Yaskawa INFORM job: DPRINT3D16.JBI

/JOB
//NAME DPRINT3D16
//POS
///NPOS 1162,0,0,0,0,0
///TOOL 9
///POSTYPE PULSE
///PULSE
C00000=35629,41672,-114626,80977,-121328,-83417,0
C00001=36190,41299,-115490,80334,-121553,-83708,0
C00002=36154,40665,-116948,80172,-121272,-84071,0
C00003=40236,36747,-126052,74955,-121987,-86900,0
C00004=40236,36690,-126053,74971,-122014,-86869,0
C00005=36377,41178,-115654,80151,-121668,-83746,0
C00006=41048,36722,-125993,74163,-122491,-86973,0
C00007=40041,36151,-127297,75001,-121635,-87147,0
C00008=35414,40629,-116901,80893,-120814,-83936,0
C00009=36299,41132,-115758,80210,-121598,-83762,0
C00010=35683,41556,-114775,80921,-121358,-83434,0
C00011=36557,42075,-113598,80267,-122151,-83252,0
C00012=42279,36667,-126139,72897,-123156,-87194,0
C00013=39910,35322,-129213,74883,-121147,-87599,0
C00014=34311,40792,-116511,81978,-120152,-83701,0
C00015=35213,41288,-115384,81279,-120939,-83528,0
C00016=34977,41570,-114734,81585,-120890,-83333,0
C00017=35446,41838,-114126,81230,-121308,-83239,0
C00018=35629,41620,-114628,80992,-121347,-83390,0
C00019=36191,41247,-115492,80349,-121573,-83680,0
C00020=36155,40612,-116951,80186,-121292,-84043,0
C00021=40236,36690,-126053,74971,-122014,-86869,0
C00022=40237,36632,-126055,74988,-122040,-86840,0
C00023=36378,41126,-115657,80166,-121688,-83719,0
C00024=41048,36664,-125996,74179,-122518,-86943,0
C00025=40042,36093,-127299,75017,-121661,-87117,0
C00026=35414,40576,-116904,80907,-120834,-83907,0
C00027=36300,41080,-115760,80225,-121617,-83734,0
C00028=35684,41505,-114777,80936,-121377,-83406,0
C00029=36558,42025,-113599,80281,-122170,-83225,0
C00030=42279,36610,-126142,72914,-123184,-87165,0
C00031=39910,35263,-129216,74898,-121175,-87568,0
C00032=34311,40739,-116513,81992,-120171,-83672,0
C00033=35213,41236,-115387,81294,-120959,-83500,0
C00034=34977,41518,-114736,81599,-120908,-83306,0
C00035=35446,41787,-114128,81244,-121328,-83211,0
C00036=35629,41569,-114630,81006,-121366,-83362,0
C00037=36191,41196,-115494,80363,-121592,-83653,0
C00038=36155,40560,-116952,80201,-121312,-84015,0
C00039=40237,36632,-126055,74988,-122040,-86840,0
C00040=40237,36575,-126058,75004,-122067,-86810,0
C00041=36378,41074,-115658,80180,-121707,-83691,0
C00042=41049,36607,-125997,74196,-122546,-86914,0
C00043=40042,36034,-127300,75033,-121689,-87086,0
C00044=35414,40524,-116905,80921,-120853,-83879,0
C00045=36300,41029,-115761,80240,-121637,-83706,0
C00046=35684,41454,-114778,80950,-121396,-83379,0
C00047=36558,41974,-113601,80296,-122190,-83197,0
C00048=42279,36552,-126143,72931,-123212,-87135,0
C00049=39911,35204,-129217,74914,-121201,-87537,0
C00050=34311,40687,-116514,82006,-120189,-83644,0
C00051=35214,41184,-115388,81308,-120977,-83472,0
C00052=34978,41467,-114738,81613,-120927,-83278,0
C00053=35447,41736,-114129,81258,-121346,-83184,0
C00054=35630,41518,-114631,81020,-121385,-83334,0
C00055=36191,41144,-115496,80378,-121612,-83625,0
C00056=36155,40507,-116953,80215,-121331,-83987,0
C00057=40237,36575,-126058,75004,-122067,-86810,0
C00058=40238,36518,-126059,75020,-122093,-86780,0
C00059=36378,41022,-115659,80195,-121727,-83663,0
C00060=41049,36550,-125999,74212,-122572,-86884,0
C00061=40042,35976,-127302,75049,-121715,-87056,0
C00062=35415,40471,-116907,80935,-120873,-83851,0
C00063=36300,40977,-115762,80254,-121657,-83679,0
C00064=35684,41402,-114780,80965,-121415,-83351,0
C00065=36558,41923,-113603,80311,-122209,-83170,0
C00066=42280,36495,-126145,72948,-123241,-87106,0
C00067=39911,35144,-129219,74930,-121229,-87507,0
C00068=34312,40635,-116515,82019,-120207,-83616,0
C00069=35214,41133,-115390,81322,-120996,-83444,0
C00070=34978,41415,-114739,81627,-120946,-83250,0
C00071=35447,41685,-114131,81273,-121365,-83157,0
C00072=35630,41466,-114633,81035,-121404,-83307,0
C00073=36192,41092,-115497,80393,-121631,-83597,0
C00074=36156,40455,-116955,80230,-121352,-83959,0
C00075=40238,36518,-126059,75020,-122093,-86780,0
C00076=40238,36460,-126060,75036,-122120,-86750,0
C00077=36379,40971,-115661,80210,-121746,-83635,0
C00078=41050,36492,-126000,74229,-122600,-86854,0
C00079=40043,35918,-127303,75065,-121742,-87026,0
C00080=35415,40419,-116908,80950,-120892,-83823,0
C00081=36301,40925,-115765,80269,-121677,-83651,0
C00082=35685,41351,-114781,80979,-121434,-83323,0
C00083=36559,41872,-113604,80326,-122228,-83142,0
C00084=42280,36438,-126146,72965,-123269,-87076,0
C00085=39912,35085,-129220,74946,-121257,-87476,0
C00086=34312,40583,-116517,82033,-120226,-83588,0
C00087=35214,41081,-115391,81336,-121015,-83416,0
C00088=34978,41364,-114741,81641,-120965,-83223,0
C00089=35447,41634,-114132,81287,-121383,-83129,0
C00090=35630,41415,-114634,81049,-121422,-83279,0
C00091=36192,41040,-115498,80408,-121651,-83569,0
C00092=36156,40403,-116956,80245,-121372,-83930,0
C00093=40238,36460,-126060,75036,-122120,-86750,0
C00094=40238,36403,-126062,75052,-122146,-86720,0
C00095=36379,40919,-115663,80225,-121767,-83607,0
C00096=41050,36435,-126001,74245,-122626,-86824,0
C00097=40043,35860,-127305,75081,-121769,-86996,0
C00098=35415,40367,-116909,80964,-120912,-83795,0
C00099=36301,40873,-115766,80284,-121697,-83623,0
C00100=35685,41300,-114783,80994,-121453,-83296,0
C00101=36559,41821,-113605,80341,-122247,-83115,0
C00102=42281,36380,-126149,72982,-123297,-87046,0
C00103=39912,35026,-129223,74962,-121284,-87445,0
C00104=34312,40531,-116519,82047,-120244,-83560,0
C00105=35215,41030,-115392,81351,-121034,-83388,0
C00106=34979,41313,-114742,81656,-120983,-83195,0
C00107=35448,41583,-114134,81302,-121401,-83101,0
C00108=35631,41364,-114636,81064,-121442,-83251,0
C00109=36192,40989,-115500,80422,-121670,-83542,0
C00110=36156,40350,-116958,80260,-121392,-83902,0
C00111=40238,36403,-126062,75052,-122146,-86720,0
C00112=40239,36346,-126064,75069,-122172,-86690,0
C00113=36379,40867,-115664,80240,-121786,-83579,0
C00114=41051,36378,-126003,74262,-122654,-86795,0
C00115=40044,35802,-127307,75097,-121796,-86965,0
C00116=35416,40315,-116910,80979,-120931,-83767,0
C00117=36301,40822,-115767,80299,-121716,-83595,0
C00118=35685,41249,-114784,81008,-121471,-83268,0
C00119=36559,41771,-113607,80356,-122267,-83088,0
C00120=42281,36323,-126150,72999,-123325,-87017,0
C00121=39912,34966,-129224,74978,-121312,-87414,0
C00122=34312,40479,-116520,82061,-120263,-83532,0
C00123=35215,40978,-115394,81365,-121052,-83361,0
C00124=34979,41262,-114744,81670,-121001,-83167,0
C00125=35448,41532,-114135,81316,-121421,-83074,0
C00126=35631,41313,-114637,81078,-121460,-83224,0
C00127=36193,40937,-115502,80437,-121690,-83514,0
C00128=36157,40298,-116959,80274,-121412,-83874,0
C00129=40239,36346,-126064,75069,-122172,-86690,0
C00130=40239,36289,-126065,75085,-122199,-86660,0
C00131=36380,40816,-115665,80255,-121806,-83551,0
C00132=41051,36321,-126004,74279,-122682,-86764,0
C00133=40044,35744,-127308,75114,-121822,-86935,0
C00134=35416,40262,-116912,80993,-120950,-83738,0
C00135=36302,40770,-115768,80314,-121736,-83567,0
C00136=35685,41197,-114785,81023,-121491,-83240,0
C00137=36560,41720,-113608,80371,-122286,-83060,0
C00138=42281,36266,-126151,73016,-123354,-86987,0
C00139=39913,34907,-129225,74994,-121339,-87383,0
C00140=34313,40427,-116521,82075,-120281,-83503,0
C00141=35215,40927,-115395,81379,-121072,-83333,0
C00142=34979,41211,-114745,81684,-121020,-83139,0
C00143=35448,41481,-114136,81331,-121439,-83046,0
C00144=35631,41262,-114638,81093,-121480,-83196,0
C00145=36193,40886,-115503,80452,-121709,-83486,0
C00146=36157,40246,-116961,80289,-121431,-83846,0
C00147=40239,36289,-126065,75085,-122199,-86660,0
C00148=40240,36231,-126066,75101,-122225,-86630,0
C00149=36380,40764,-115666,80270,-121825,-83524,0
C00150=41051,36264,-126005,74295,-122708,-86735,0
C00151=40044,35686,-127309,75130,-121850,-86905,0
C00152=35416,40210,-116913,81007,-120969,-83710,0
C00153=36302,40718,-115769,80329,-121755,-83539,0
C00154=35686,41146,-114787,81037,-121511,-83212,0
C00155=36560,41669,-113609,80387,-122306,-83033,0
C00156=42282,36209,-126152,73033,-123383,-86957,0
C00157=39913,34848,-129226,75010,-121367,-87352,0
C00158=34313,40375,-116522,82089,-120299,-83475,0
C00159=35216,40875,-115396,81394,-121090,-83305,0
C00160=34980,41159,-114746,81698,-121038,-83112,0
C00161=35449,41430,-114137,81345,-121458,-83019,0
C00162=35632,41210,-114639,81108,-121498,-83168,0
C00163=36193,40834,-115504,80467,-121729,-83458,0
C00164=36157,40194,-116962,80304,-121452,-83818,0
C00165=40240,36231,-126066,75101,-122225,-86630,0
C00166=40240,36174,-126067,75118,-122252,-86600,0
C00167=36380,40713,-115667,80285,-121845,-83495,0
C00168=41052,36207,-126006,74312,-122736,-86705,0
C00169=40045,35629,-127310,75146,-121876,-86874,0
C00170=35417,40158,-116914,81022,-120989,-83682,0
C00171=36302,40667,-115771,80344,-121775,-83511,0
C00172=35686,41095,-114788,81052,-121529,-83184,0
C00173=36560,41619,-113610,80402,-122324,-83005,0
C00174=42282,36152,-126153,73051,-123410,-86927,0
C00175=39914,34789,-129227,75027,-121394,-87321,0
C00176=34314,40323,-116523,82102,-120318,-83447,0
C00177=35216,40824,-115397,81408,-121110,-83276,0
C00178=34980,41108,-114747,81713,-121057,-83084,0
C00179=35449,41379,-114138,81360,-121476,-82991,0
C00180=35632,41159,-114640,81122,-121517,-83141,0
C00181=36194,40783,-115505,80482,-121748,-83430,0
C00182=36158,40142,-116962,80319,-121471,-83789,0
C00183=40240,36174,-126067,75118,-122252,-86600,0
C00184=40240,36117,-126068,75134,-122278,-86570,0
C00185=36381,40661,-115668,80300,-121866,-83467,0
C00186=41052,36150,-126007,74329,-122763,-86674,0
C00187=40045,35571,-127311,75162,-121902,-86844,0
C00188=35417,40106,-116915,81036,-121008,-83654,0
C00189=36303,40615,-115772,80359,-121796,-83483,0
C00190=35687,41044,-114789,81067,-121548,-83156,0
C00191=36561,41568,-113611,80417,-122344,-82978,0
C00192=42283,36095,-126154,73068,-123439,-86897,0
C00193=39914,34730,-129228,75043,-121422,-87290,0
C00194=34314,40271,-116524,82116,-120336,-83419,0
C00195=35216,40773,-115398,81422,-121128,-83249,0
C00196=34980,41057,-114748,81727,-121075,-83056,0
C00197=35449,41328,-114139,81374,-121496,-82963,0
C00198=35632,41108,-114641,81137,-121536,-83113,0
C00199=36194,40732,-115506,80497,-121768,-83402,0
C00200=36158,40089,-116963,80334,-121492,-83761,0
C00201=40240,36117,-126068,75134,-122278,-86570,0
C00202=40241,36060,-126069,75151,-122305,-86540,0
C00203=36381,40610,-115669,80315,-121885,-83439,0
C00204=41053,36093,-126008,74346,-122790,-86645,0
C00205=40046,35513,-127313,75179,-121930,-86813,0
C00206=35417,40054,-116916,81051,-121028,-83625,0
C00207=36303,40564,-115773,80374,-121815,-83455,0
C00208=35687,40993,-114789,81082,-121567,-83128,0
C00209=36561,41518,-113612,80432,-122363,-82950,0
C00210=42283,36037,-126155,73085,-123468,-86868,0
C00211=39914,34671,-129229,75059,-121450,-87259,0
C00212=34314,40219,-116526,82130,-120355,-83390,0
C00213=35217,40721,-115399,81437,-121146,-83221,0
C00214=34981,41006,-114749,81741,-121093,-83028,0
C00215=35449,41278,-114140,81389,-121514,-82935,0
C00216=35633,41057,-114642,81152,-121555,-83085,0
C00217=36194,40680,-115506,80512,-121788,-83374,0
C00218=36158,40037,-116964,80348,-121512,-83733,0
C00219=40241,36060,-126069,75151,-122305,-86540,0
C00220=40241,36003,-126069,75167,-122331,-86510,0
C00221=36381,40558,-115669,80330,-121905,-83412,0
C00222=41053,36036,-126010,74363,-122817,-86615,0
C00223=40046,35455,-127313,75195,-121956,-86783,0
C00224=35418,40002,-116917,81065,-121047,-83597,0
C00225=36303,40512,-115773,80389,-121835,-83427,0
C00226=35687,40942,-114790,81096,-121586,-83101,0
C00227=36561,41467,-113613,80447,-122383,-82922,0
C00228=42284,35980,-126155,73103,-123495,-86837,0
C00229=39915,34612,-129229,75075,-121477,-87228,0
C00230=34314,40167,-116526,82144,-120373,-83362,0
C00231=35217,40670,-115400,81451,-121166,-83193,0
C00232=34981,40955,-114750,81756,-121112,-83000,0
C00233=35450,41227,-114141,81404,-121532,-82907,0
C00234=35633,41006,-114643,81166,-121574,-83057,0
C00235=36195,40629,-115507,80527,-121807,-83346,0
C00236=36159,39985,-116966,80363,-121531,-83705,0
C00237=40241,36003,-126069,75167,-122331,-86510,0
C00238=40242,35946,-126070,75184,-122357,-86479,0
C00239=36382,40507,-115671,80345,-121924,-83383,0
C00240=41053,35979,-126011,74380,-122845,-86584,0
C00241=40046,35397,-127314,75212,-121983,-86752,0
C00242=35418,39950,-116917,81080,-121067,-83568,0
C00243=36304,40461,-115774,80404,-121854,-83399,0
C00244=35688,40891,-114791,81111,-121605,-83073,0
C00245=36562,41417,-113614,80462,-122402,-82895,0
C00246=42284,35923,-126157,73120,-123524,-86808,0
C00247=39915,34553,-129231,75092,-121505,-87197,0
C00248=34315,40116,-116527,82158,-120391,-83333,0
C00249=35217,40619,-115400,81466,-121184,-83164,0
C00250=34981,40904,-114750,81770,-121130,-82972,0
C00251=35450,41176,-114142,81418,-121551,-82880,0
C00252=35633,40956,-114644,81181,-121593,-83029,0
C00253=36195,40577,-115509,80542,-121827,-83318,0
C00254=36159,39933,-116966,80378,-121552,-83676,0
C00255=40242,35946,-126070,75184,-122357,-86479,0
C00256=40242,35889,-126072,75200,-122385,-86449,0
C00257=36382,40456,-115672,80360,-121945,-83355,0
C00258=41054,35922,-126011,74397,-122871,-86554,0
C00259=40047,35340,-127315,75228,-122010,-86721,0
C00260=35418,39898,-116919,81095,-121087,-83540,0
C00261=36304,40409,-115775,80419,-121874,-83370,0
C00262=35688,40840,-114792,81126,-121624,-83045,0
C00263=36562,41366,-113614,80478,-122421,-82867,0
C00264=42284,35866,-126158,73137,-123553,-86778,0
C00265=39916,34494,-129232,75108,-121532,-87165,0
C00266=34315,40064,-116528,82172,-120410,-83305,0
C00267=35218,40567,-115402,81481,-121203,-83137,0
C00268=34982,40853,-114751,81784,-121149,-82944,0
C00269=35450,41126,-114142,81433,-121569,-82852,0
C00270=35634,40905,-114644,81196,-121612,-83001,0
C00271=36195,40526,-115509,80557,-121846,-83290,0
C00272=36159,39881,-116967,80393,-121571,-83648,0
C00273=40242,35889,-126072,75200,-122385,-86449,0
C00274=40242,35833,-126072,75217,-122411,-86419,0
C00275=36383,40404,-115672,80375,-121964,-83327,0
C00276=41054,35865,-126012,74413,-122899,-86524,0
C00277=40047,35282,-127315,75245,-122037,-86691,0
C00278=35419,39846,-116919,81109,-121105,-83511,0
C00279=36304,40358,-115775,80434,-121894,-83343,0
C00280=35688,40789,-114792,81141,-121643,-83017,0
C00281=36562,41316,-113615,80493,-122440,-82839,0
C00282=42285,35809,-126158,73155,-123580,-86748,0
C00283=39916,34435,-129232,75124,-121560,-87135,0
C00284=34315,40012,-116528,82187,-120428,-83277,0
C00285=35218,40516,-115402,81495,-121222,-83108,0
C00286=34982,40803,-114752,81799,-121167,-82916,0
C00287=35451,41075,-114143,81448,-121589,-82824,0
C00288=35634,40854,-114645,81211,-121630,-82973,0
C00289=36196,40475,-115510,80572,-121866,-83262,0
C00290=36160,39830,-116968,80408,-121592,-83619,0
C00291=40242,35833,-126072,75217,-122411,-86419,0
C00292=40243,35776,-126072,75234,-122438,-86388,0
C00293=36383,40353,-115672,80390,-121984,-83299,0
C00294=41055,35808,-126012,74431,-122926,-86495,0
C00295=40048,35224,-127315,75261,-122063,-86661,0
C00296=35419,39794,-116920,81124,-121124,-83483,0
C00297=36305,40307,-115775,80449,-121914,-83314,0
C00298=35688,40738,-114793,81156,-121662,-82989,0
C00299=36563,41266,-113615,80508,-122460,-82812,0
C00300=42285,35753,-126158,73172,-123609,-86718,0
C00301=39917,34376,-129233,75141,-121588,-87103,0
C00302=34316,39960,-116528,82201,-120446,-83248,0
C00303=35218,40465,-115403,81510,-121241,-83080,0
C00304=34982,40752,-114752,81813,-121185,-82888,0
C00305=35451,41024,-114143,81462,-121607,-82797,0
C00306=35634,40803,-114646,81226,-121650,-82945,0
C00307=36196,40424,-115510,80587,-121885,-83234,0
C00308=36160,39778,-116968,80423,-121612,-83591,0
C00309=40243,35776,-126072,75234,-122438,-86388,0
C00310=40243,35719,-126073,75250,-122464,-86358,0
C00311=36383,40302,-115673,80406,-122004,-83271,0
C00312=41055,35751,-126012,74448,-122953,-86464,0
C00313=40048,35167,-127316,75278,-122091,-86630,0
C00314=35419,39743,-116920,81139,-121144,-83455,0
C00315=36305,40255,-115776,80464,-121933,-83286,0
C00316=35689,40687,-114793,81170,-121681,-82961,0
C00317=36563,41215,-113616,80524,-122479,-82784,0
C00318=42286,35696,-126159,73190,-123638,-86688,0
C00319=39917,34317,-129233,75157,-121615,-87072,0
C00320=34316,39909,-116529,82215,-120465,-83220,0
C00321=35219,40414,-115403,81524,-121260,-83052,0
C00322=34983,40701,-114752,81828,-121204,-82860,0
C00323=35451,40974,-114144,81477,-121625,-82769,0
C00324=35635,40752,-114646,81240,-121668,-82917,0
C00325=36196,40373,-115511,80602,-121905,-83206,0
C00326=36161,39726,-116968,80438,-121631,-83562,0
C00327=40243,35719,-126073,75250,-122464,-86358,0
C00328=40244,35662,-126073,75267,-122491,-86328,0
C00329=36383,40251,-115673,80421,-122023,-83243,0
C00330=41055,35695,-126013,74465,-122980,-86434,0
C00331=40049,35109,-127316,75294,-122117,-86599,0
C00332=35420,39691,-116920,81153,-121164,-83426,0
C00333=36306,40204,-115776,80480,-121953,-83258,0
C00334=35689,40637,-114793,81185,-121700,-82933,0
C00335=36563,41165,-113616,80539,-122499,-82756,0
C00336=42286,35639,-126159,73208,-123665,-86658,0
C00337=39917,34258,-129233,75174,-121643,-87041,0
C00338=34316,39857,-116529,82229,-120483,-83191,0
C00339=35219,40363,-115403,81539,-121278,-83024,0
C00340=34983,40650,-114753,81843,-121222,-82832,0
C00341=35452,40923,-114144,81492,-121644,-82741,0
C00342=35635,40702,-114646,81255,-121688,-82889,0
C00343=36197,40322,-115511,80617,-121925,-83178,0
C00344=36161,39674,-116969,80454,-121652,-83534,0
C00345=40244,35662,-126073,75267,-122491,-86328,0
C00346=40244,35605,-126073,75284,-122517,-86298,0
C00347=36384,40199,-115673,80436,-122044,-83214,0
C00348=41056,35638,-126013,74482,-123008,-86403,0
C00349=40049,35052,-127316,75311,-122145,-86568,0
C00350=35420,39639,-116920,81168,-121183,-83398,0
C00351=36306,40153,-115776,80495,-121973,-83230,0
C00352=35689,40586,-114794,81200,-121719,-82905,0
C00353=36564,41115,-113616,80555,-122518,-82729,0
C00354=42286,35582,-126159,73225,-123694,-86628,0
C00355=39918,34200,-129234,75190,-121670,-87009,0
C00356=34317,39806,-116529,82243,-120502,-83163,0
C00357=35219,40312,-115404,81554,-121297,-82996,0
C00358=34983,40599,-114753,81857,-121241,-82804,0
C00359=35452,40873,-114144,81507,-121663,-82712,0
C00360=35635,40651,-114647,81270,-121706,-82861,0
C00361=36197,40270,-115511,80632,-121945,-83149,0
C00362=36161,39622,-116969,80469,-121671,-83506,0
C00363=40244,35605,-126073,75284,-122517,-86298,0
C00364=40244,35549,-126073,75301,-122544,-86267,0
C00365=36384,40148,-115673,80451,-122063,-83186,0
C00366=41056,35581,-126013,74499,-123034,-86373,0
C00367=40049,34994,-127317,75328,-122171,-86537,0
C00368=35420,39587,-116921,81183,-121203,-83369,0
C00369=36306,40102,-115776,80510,-121993,-83202,0
C00370=35690,40535,-114794,81215,-121738,-82877,0
C00371=36564,41065,-113616,80570,-122537,-82701,0
C00372=42287,35525,-126159,73243,-123723,-86598,0
C00373=39918,34141,-129234,75207,-121698,-86978,0
C00374=34317,39754,-116529,82257,-120520,-83134,0
C00375=35220,40261,-115404,81569,-121316,-82967,0
C00376=34984,40549,-114753,81872,-121260,-82776,0
C00377=35452,40822,-114144,81522,-121682,-82685,0
C00378=35636,40600,-114647,81285,-121725,-82833,0
C00379=36197,40219,-115511,80648,-121964,-83121,0
C00380=36162,39570,-116969,80484,-121692,-83477,0
C00381=40244,35549,-126073,75301,-122544,-86267,0
C00382=40245,35492,-126074,75318,-122570,-86237,0
C00383=36384,40097,-115673,80467,-122083,-83158,0
C00384=41057,35525,-126013,74516,-123062,-86343,0
C00385=40050,34937,-127317,75344,-122198,-86507,0
C00386=35421,39536,-116921,81198,-121222,-83340,0
C00387=36307,40051,-115776,80525,-122013,-83173,0
C00388=35690,40484,-114794,81230,-121758,-82849,0
C00389=36564,41015,-113616,80586,-122556,-82673,0
C00390=42287,35469,-126160,73261,-123750,-86568,0
C00391=39919,34082,-129234,75223,-121725,-86947,0
C00392=34317,39703,-116530,82272,-120538,-83106,0
C00393=35220,40210,-115404,81583,-121335,-82939,0
C00394=34984,40498,-114753,81886,-121278,-82748,0
C00395=35453,40772,-114145,81537,-121700,-82657,0
C00396=35636,40550,-114647,81300,-121744,-82805,0
C00397=36198,40168,-115511,80663,-121984,-83093,0
C00398=36162,39519,-116969,80499,-121712,-83449,0
C00399=40245,35492,-126074,75318,-122570,-86237,0
C00400=40245,35435,-126074,75335,-122597,-86206,0
C00401=36385,40046,-115673,80482,-122102,-83130,0
C00402=41057,35468,-126013,74534,-123089,-86313,0
C00403=40050,34879,-127317,75361,-122225,-86476,0
C00404=35421,39484,-116921,81213,-121242,-83312,0
C00405=36307,40000,-115776,80541,-122032,-83145,0
C00406=35690,40434,-114794,81245,-121776,-82820,0
C00407=36565,40965,-113616,80601,-122576,-82645,0
C00408=42288,35412,-126160,73279,-123779,-86537,0
C00409=39919,34024,-129234,75240,-121753,-86915,0
C00410=34318,39651,-116529,82286,-120557,-83077,0
C00411=35220,40159,-115404,81598,-121353,-82911,0
C00412=34984,40447,-114753,81901,-121297,-82719,0
C00413=35453,40722,-114145,81552,-121719,-82629,0
C00414=35636,40499,-114647,81315,-121763,-82777,0
C00415=36198,40117,-115511,80678,-122004,-83065,0
C00416=36162,39467,-116969,80514,-121731,-83420,0
C00417=40245,35435,-126074,75335,-122597,-86206,0
C00418=40246,35379,-126073,75352,-122623,-86176,0
C00419=36385,39995,-115673,80498,-122123,-83101,0
C00420=41057,35412,-126013,74551,-123116,-86283,0
C00421=40051,34822,-127316,75378,-122252,-86445,0
C00422=35421,39432,-116921,81228,-121261,-83283,0
C00423=36307,39948,-115776,80556,-122052,-83116,0
C00424=35691,40383,-114794,81260,-121796,-82792,0
C00425=36565,40914,-113616,80617,-122595,-82617,0
C00426=42288,35355,-126159,73296,-123808,-86507,0
C00427=39920,33965,-129234,75257,-121781,-86884,0
C00428=34318,39600,-116529,82300,-120575,-83048,0
C00429=35220,40108,-115404,81613,-121373,-82882,0
C00430=34985,40397,-114753,81916,-121315,-82691,0
C00431=35453,40671,-114144,81566,-121738,-82600,0
C00432=35637,40449,-114647,81330,-121782,-82749,0
C00433=36198,40066,-115511,80694,-122023,-83036,0
C00434=36163,39415,-116969,80530,-121752,-83391,0
C00435=40246,35379,-126073,75352,-122623,-86176,0
C00436=40246,35322,-126073,75369,-122649,-86145,0
C00437=36385,39944,-115673,80513,-122143,-83073,0
C00438=41058,35355,-126013,74568,-123144,-86252,0
C00439=40051,34765,-127316,75395,-122279,-86414,0
C00440=35422,39381,-116920,81243,-121280,-83254,0
C00441=36308,39897,-115776,80571,-122071,-83088,0
C00442=35691,40333,-114794,81276,-121814,-82764,0
C00443=36565,40864,-113616,80632,-122615,-82589,0
C00444=42289,35299,-126159,73314,-123835,-86477,0
C00445=39920,33906,-129233,75274,-121808,-86853,0
C00446=34318,39548,-116529,82315,-120595,-83020,0
C00447=35221,40057,-115403,81628,-121391,-82854,0
C00448=34985,40346,-114753,81931,-121334,-82663,0
C00449=35454,40621,-114144,81582,-121756,-82573,0
C00450=35637,40398,-114646,81345,-121801,-82720,0
C00451=36199,40016,-115511,80709,-122043,-83008,0
C00452=36163,39364,-116969,80545,-121771,-83363,0
C00453=40246,35322,-126073,75369,-122649,-86145,0
C00454=40246,35266,-126073,75386,-122677,-86115,0
C00455=36386,39893,-115673,80529,-122162,-83045,0
C00456=41058,35299,-126013,74586,-123171,-86222,0
C00457=40052,34708,-127316,75412,-122306,-86383,0
C00458=35422,39329,-116920,81257,-121299,-83225,0
C00459=36308,39847,-115776,80587,-122092,-83060,0
C00460=35691,40282,-114793,81291,-121833,-82736,0
C00461=36566,40814,-113616,80648,-122634,-82562,0
C00462=42289,35242,-126159,73332,-123864,-86446,0
C00463=39920,33848,-129233,75290,-121836,-86821,0
C00464=34319,39497,-116529,82329,-120613,-82991,0
C00465=35221,40006,-115403,81643,-121411,-82826,0
C00466=34985,40296,-114753,81945,-121352,-82635,0
C00467=35454,40571,-114144,81596,-121775,-82545,0
C00468=35637,40348,-114646,81360,-121820,-82693,0
C00469=36199,39965,-115511,80724,-122062,-82980,0
C00470=36163,39312,-116968,80560,-121792,-83334,0
C00471=40246,35266,-126073,75386,-122677,-86115,0
C00472=40247,35209,-126073,75403,-122703,-86084,0
C00473=36386,39842,-115673,80544,-122182,-83016,0
C00474=41059,35242,-126012,74603,-123199,-86191,0
C00475=40052,34650,-127316,75429,-122332,-86352,0
C00476=35422,39278,-116920,81272,-121319,-83197,0
C00477=36308,39796,-115776,80602,-122112,-83032,0
C00478=35692,40232,-114793,81306,-121852,-82708,0
C00479=36566,40764,-113616,80664,-122653,-82534,0
C00480=42289,35186,-126159,73350,-123893,-86416,0
C00481=39921,33790,-129233,75307,-121863,-86789,0
C00482=34319,39446,-116529,82343,-120631,-82962,0
C00483=35222,39956,-115403,81657,-121429,-82797,0
C00484=34985,40245,-114752,81960,-121370,-82607,0
C00485=35454,40521,-114144,81612,-121793,-82516,0
C00486=35638,40297,-114646,81376,-121839,-82664,0
C00487=36199,39914,-115510,80740,-122082,-82951,0
C00488=36164,39261,-116968,80576,-121812,-83305,0
C00489=40247,35209,-126073,75403,-122703,-86084,0
C00490=40247,35153,-126072,75420,-122730,-86054,0
C00491=36387,39792,-115672,80560,-122201,-82988,0
C00492=41059,35186,-126012,74621,-123225,-86161,0
C00493=40052,34593,-127315,75446,-122360,-86322,0
C00494=35423,39226,-116919,81287,-121338,-83168,0
C00495=36308,39745,-115775,80618,-122131,-83003,0
C00496=35692,40181,-114793,81321,-121871,-82679,0
C00497=36566,40715,-113615,80679,-122672,-82506,0
C00498=42290,35129,-126158,73368,-123920,-86386,0
C00499=39921,33731,-129232,75324,-121891,-86758,0
C00500=34319,39395,-116528,82358,-120650,-82933,0
C00501=35222,39905,-115403,81672,-121447,-82769,0
C00502=34986,40195,-114752,81975,-121389,-82578,0
C00503=35455,40471,-114143,81627,-121813,-82488,0
C00504=35638,40247,-114645,81391,-121858,-82636,0
C00505=36200,39863,-115510,80755,-122101,-82923,0
C00506=36164,39209,-116968,80591,-121831,-83276,0
C00507=40247,35153,-126072,75420,-122730,-86054,0
C00508=40248,35097,-126072,75437,-122756,-86023,0
C00509=36387,39741,-115672,80575,-122222,-82960,0
C00510=41060,35130,-126011,74638,-123253,-86130,0
C00511=40053,34536,-127315,75463,-122386,-86290,0
C00512=35423,39175,-116919,81303,-121358,-83139,0
C00513=36309,39694,-115775,80633,-122151,-82975,0
C00514=35692,40131,-114792,81336,-121890,-82651,0
C00515=36567,40665,-113615,80695,-122692,-82477,0
C00516=42290,35073,-126158,73386,-123949,-86356,0
C00517=39922,33673,-129232,75341,-121919,-86727,0
C00518=34320,39343,-116528,82372,-120668,-82905,0
C00519=35222,39854,-115402,81687,-121467,-82740,0
C00520=34986,40144,-114751,81990,-121407,-82550,0
C00521=35455,40420,-114143,81642,-121831,-82460,0
C00522=35638,40196,-114645,81406,-121877,-82608,0
C00523=36200,39812,-115510,80771,-122121,-82895,0
C00524=36164,39158,-116967,80606,-121852,-83248,0
C00525=40248,35097,-126072,75437,-122756,-86023,0
C00526=40248,35040,-126070,75454,-122783,-85993,0
C00527=36387,39690,-115671,80591,-122241,-82931,0
C00528=41060,35073,-126011,74656,-123280,-86100,0
C00529=40053,34479,-127314,75480,-122414,-86260,0
C00530=35423,39123,-116919,81318,-121377,-83110,0
C00531=36309,39643,-115774,80649,-122170,-82946,0
C00532=35693,40080,-114791,81351,-121909,-82623,0
C00533=36567,40615,-113614,80711,-122711,-82450,0
C00534=42291,35016,-126157,73404,-123978,-86325,0
C00535=39922,33614,-129231,75358,-121946,-86695,0
C00536=34320,39292,-116527,82387,-120687,-82876,0
C00537=35223,39803,-115402,81702,-121485,-82712,0
C00538=34986,40094,-114751,82005,-121426,-82521,0
C00539=35455,40370,-114142,81657,-121850,-82432,0
C00540=35639,40146,-114644,81421,-121896,-82579,0
C00541=36200,39762,-115509,80786,-122140,-82866,0
C00542=36165,39106,-116967,80622,-121871,-83219,0
C00543=40248,35040,-126070,75454,-122783,-85993,0
C00544=40249,34984,-126070,75471,-122809,-85962,0
C00545=36388,39639,-115671,80606,-122261,-82903,0
C00546=41060,35017,-126010,74673,-123307,-86069,0
C00547=40054,34422,-127314,75497,-122440,-86228,0
C00548=35424,39072,-116917,81333,-121397,-83082,0
C00549=36310,39592,-115774,80665,-122191,-82917,0
C00550=35693,40030,-114791,81367,-121929,-82595,0
C00551=36567,40565,-113613,80726,-122731,-82422,0
C00552=42291,34960,-126157,73422,-124007,-86295,0
C00553=39922,33556,-129231,75375,-121974,-86663,0
C00554=34320,39241,-116527,82401,-120705,-82848,0
C00555=35223,39753,-115400,81717,-121505,-82683,0
C00556=34987,40044,-114750,82019,-121444,-82494,0
C00557=35456,40320,-114141,81672,-121868,-82404,0
C00558=35639,40096,-114644,81436,-121915,-82551,0
C00559=36201,39711,-115509,80802,-122160,-82838,0
C00560=36165,39055,-116966,80637,-121892,-83191,0
C00561=40249,34984,-126070,75471,-122809,-85962,0
C00562=40249,34928,-126069,75489,-122836,-85931,0
C00563=36388,39588,-115669,80622,-122280,-82874,0
C00564=41061,34961,-126010,74691,-123334,-86039,0
C00565=40054,34365,-127313,75514,-122467,-86197,0
C00566=35424,39021,-116916,81348,-121416,-83053,0
C00567=36310,39541,-115773,80680,-122210,-82889,0
C00568=35693,39980,-114790,81382,-121947,-82566,0
C00569=36568,40515,-113613,80742,-122750,-82393,0
C00570=42292,34904,-126155,73440,-124034,-86264,0
C00571=39923,33498,-129229,75392,-122001,-86631,0
C00572=34321,39190,-116526,82416,-120723,-82819,0
C00573=35223,39702,-115399,81732,-121523,-82655,0
C00574=34987,39993,-114749,82034,-121462,-82465,0
C00575=35456,40270,-114141,81687,-121887,-82375,0
C00576=35639,40046,-114643,81452,-121933,-82523,0
C00577=36201,39660,-115507,80817,-122179,-82809,0
C00578=36165,39004,-116966,80653,-121912,-83161,0
C00579=40249,34928,-126069,75489,-122836,-85931,0
C00580=40249,34871,-126068,75506,-122862,-85900,0
C00581=36388,39538,-115668,80638,-122301,-82845,0
C00582=41061,34905,-126008,74709,-123362,-86008,0
C00583=40054,34308,-127311,75531,-122494,-86166,0
C00584=35424,38970,-116916,81363,-121436,-83024,0
C00585=36310,39491,-115772,80696,-122230,-82860,0
C00586=35694,39929,-114789,81397,-121967,-82538,0
C00587=36568,40465,-113612,80758,-122770,-82365,0
C00588=42292,34847,-126154,73459,-124063,-86234,0
C00589=39923,33440,-129228,75409,-122029,-86600,0
C00590=34321,39139,-116524,82430,-120742,-82790,0
C00591=35223,39652,-115399,81747,-121542,-82626,0
C00592=34987,39943,-114749,82049,-121482,-82437,0
C00593=35456,40220,-114140,81702,-121906,-82347,0
C00594=35640,39995,-114642,81467,-121953,-82494,0
C00595=36201,39610,-115506,80833,-122199,-82781,0
C00596=36166,38952,-116964,80668,-121932,-83132,0
C00597=40249,34871,-126068,75506,-122862,-85900,0
C00598=40250,34815,-126067,75523,-122890,-85870,0
C00599=36389,39487,-115668,80653,-122321,-82817,0
C00600=41062,34848,-126007,74726,-123389,-85978,0
C00601=40055,34251,-127310,75549,-122521,-86135,0
C00602=35425,38918,-116915,81378,-121455,-82995,0
C00603=36311,39440,-115772,80711,-122249,-82832,0
C00604=35694,39879,-114788,81413,-121985,-82509,0
C00605=36568,40416,-113611,80774,-122788,-82338,0
C00606=42292,34791,-126153,73477,-124092,-86203,0
C00607=39924,33381,-129228,75426,-122056,-86568,0
C00608=34321,39088,-116524,82445,-120760,-82761,0
C00609=35224,39601,-115398,81763,-121561,-82598,0
C00610=34988,39893,-114748,82064,-121500,-82408,0
C00611=35457,40170,-114139,81718,-121924,-82319,0
C00612=35640,39945,-114641,81482,-121971,-82466,0
C00613=36202,39559,-115505,80848,-122220,-82752,0
C00614=36166,38901,-116963,80684,-121952,-83104,0
C00615=40250,34815,-126067,75523,-122890,-85870,0
C00616=40250,34759,-126067,75541,-122916,-85839,0
C00617=36389,39436,-115667,80669,-122340,-82788,0
C00618=41062,34792,-126006,74744,-123416,-85947,0
C00619=40055,34194,-127309,75566,-122548,-86104,0
C00620=35425,38867,-116914,81393,-121475,-82966,0
C00621=36311,39389,-115771,80727,-122270,-82803,0
C00622=35694,39829,-114787,81428,-122005,-82481,0
C00623=36569,40366,-113610,80790,-122808,-82309,0
C00624=42293,34735,-126152,73495,-124119,-86173,0
C00625=39924,33323,-129227,75443,-122084,-86536,0
C00626=34322,39037,-116523,82460,-120779,-82732,0
C00627=35224,39551,-115397,81778,-121580,-82569,0
C00628=34988,39843,-114747,82079,-121519,-82380,0
C00629=35457,40120,-114138,81733,-121943,-82291,0
C00630=35640,39895,-114640,81498,-121991,-82438,0
C00631=36202,39509,-115504,80864,-122239,-82723,0
C00632=36166,38850,-116962,80700,-121971,-83075,0
C00633=40250,34759,-126067,75541,-122916,-85839,0
C00634=40251,34703,-126066,75558,-122942,-85808,0
C00635=36389,39386,-115666,80685,-122360,-82760,0
C00636=41063,34736,-126005,74762,-123443,-85916,0
C00637=40056,34137,-127308,75583,-122575,-86073,0
C00638=35425,38816,-116913,81409,-121493,-82938,0
C00639=36311,39339,-115769,80743,-122290,-82774,0
C00640=35695,39779,-114786,81444,-122023,-82452,0
C00641=36569,40316,-113609,80806,-122827,-82281,0
C00642=42293,34679,-126152,73514,-124148,-86142,0
C00643=39925,33265,-129226,75461,-122112,-86505,0
C00644=34322,38986,-116522,82474,-120797,-82703,0
C00645=35224,39500,-115396,81793,-121599,-82541,0
C00646=34988,39793,-114745,82094,-121537,-82351,0
C00647=35457,40071,-114137,81748,-121962,-82262,0
C00648=35641,39845,-114639,81513,-122009,-82409,0
C00649=36202,39458,-115503,80880,-122259,-82695,0
C00650=36167,38799,-116961,80715,-121992,-83046,0
C00651=40251,34703,-126066,75558,-122942,-85808,0
C00652=40251,34647,-126064,75576,-122969,-85777,0
C00653=36390,39335,-115665,80701,-122380,-82731,0
C00654=41063,34680,-126004,74780,-123471,-85885,0
C00655=40056,34080,-127307,75601,-122602,-86042,0
C00656=35426,38765,-116912,81424,-121513,-82909,0
C00657=36312,39288,-115768,80759,-122309,-82746,0
C00658=35695,39729,-114785,81459,-122043,-82424,0
C00659=36569,40267,-113608,80822,-122847,-82253,0
C00660=42294,34623,-126150,73532,-124177,-86112,0
C00661=39925,33207,-129224,75478,-122139,-86473,0
C00662=34322,38935,-116521,82489,-120815,-82674,0
C00663=35225,39450,-115395,81808,-121617,-82512,0
C00664=34989,39743,-114744,82110,-121555,-82322,0
C00665=35458,40021,-114136,81764,-121981,-82234,0
C00666=35641,39795,-114638,81529,-122029,-82381,0
C00667=36203,39408,-115502,80895,-122278,-82667,0
C00668=36167,38748,-116960,80731,-122012,-83017,0
C00669=40251,34647,-126064,75576,-122969,-85777,0
C00670=40251,34591,-126062,75593,-122995,-85747,0
C00671=36390,39285,-115664,80717,-122400,-82703,0
C00672=41063,34624,-126003,74798,-123499,-85855,0
C00673=40056,34023,-127306,75618,-122629,-86011,0
C00674=35426,38714,-116910,81439,-121532,-82879,0
C00675=36312,39238,-115767,80774,-122329,-82717,0
C00676=35695,39679,-114784,81475,-122062,-82396,0
C00677=36569,40217,-113606,80838,-122867,-82224,0
C00678=42294,34567,-126149,73550,-124205,-86081,0
C00679=39925,33149,-129223,75495,-122167,-86441,0
C00680=34323,38884,-116520,82504,-120834,-82645,0
C00681=35225,39400,-115394,81823,-121636,-82483,0
C00682=34989,39692,-114743,82125,-121574,-82294,0
C00683=35458,39971,-114134,81779,-121999,-82205,0
C00684=35641,39745,-114637,81544,-122047,-82352,0
C00685=36203,39357,-115500,80911,-122298,-82638,0
C00686=36167,38697,-116959,80747,-122032,-82988,0
C00687=40251,34591,-126062,75593,-122995,-85747,0
C00688=40252,34535,-126061,75611,-123022,-85716,0
C00689=36390,39234,-115661,80732,-122420,-82673,0
C00690=41064,34568,-126001,74815,-123525,-85824,0
C00691=40057,33967,-127305,75635,-122655,-85979,0
C00692=35426,38663,-116909,81454,-121552,-82850,0
C00693=36312,39187,-115765,80790,-122348,-82689,0
C00694=35696,39629,-114782,81490,-122081,-82367,0
C00695=36570,40168,-113605,80854,-122886,-82197,0
C00696=42295,34511,-126147,73569,-124233,-86051,0
C00697=39926,33091,-129221,75513,-122194,-86409,0
C00698=34323,38833,-116517,82518,-120852,-82616,0
C00699=35225,39349,-115392,81839,-121655,-82455,0
C00700=34989,39642,-114742,82140,-121592,-82266,0
C00701=35458,39921,-114133,81794,-122017,-82177,0
C00702=35641,39695,-114635,81559,-122067,-82324,0
C00703=36203,39307,-115499,80927,-122317,-82609,0
C00704=36168,38645,-116958,80762,-122052,-82959,0
C00705=40252,34535,-126061,75611,-123022,-85716,0
C00706=40252,34479,-126060,75628,-123048,-85685,0
C00707=36391,39184,-115660,80748,-122439,-82645,0
C00708=41064,34512,-125999,74833,-123553,-85793,0
C00709=40057,33910,-127303,75653,-122683,-85948,0
C00710=35427,38612,-116907,81470,-121571,-82821,0
C00711=36313,39137,-115764,80806,-122369,-82660,0
C00712=35696,39579,-114781,81506,-122100,-82338,0
C00713=36570,40118,-113604,80870,-122904,-82168,0
C00714=42295,34455,-126146,73587,-124262,-86020,0
C00715=39926,33033,-129220,75530,-122222,-86377,0
C00716=34323,38782,-116516,82533,-120872,-82587,0
C00717=35226,39299,-115390,81854,-121674,-82426,0
C00718=34990,39592,-114740,82155,-121611,-82237,0
C00719=35459,39871,-114132,81810,-122037,-82148,0
C00720=35642,39645,-114634,81575,-122085,-82295,0
C00721=36204,39256,-115498,80943,-122337,-82581,0
C00722=36168,38594,-116956,80778,-122072,-82930,0
C00723=40252,34479,-126060,75628,-123048,-85685,0
C00724=40253,34423,-126058,75646,-123075,-85654,0
C00725=36391,39134,-115659,80764,-122460,-82616,0
C00726=41065,34456,-125998,74851,-123580,-85762,0
C00727=40058,33853,-127301,75671,-122709,-85917,0
C00728=35427,38561,-116906,81485,-121591,-82792,0
C00729=36313,39086,-115762,80822,-122389,-82631,0
C00730=35696,39529,-114779,81521,-122118,-82310,0
C00731=36571,40069,-113602,80886,-122924,-82140,0
C00732=42295,34399,-126144,73606,-124290,-85989,0
C00733=39927,32975,-129218,75547,-122249,-86345,0
C00734=34324,38731,-116515,82548,-120890,-82558,0
C00735=35226,39249,-115389,81869,-121693,-82397,0
C00736=34990,39542,-114739,82170,-121629,-82208,0
C00737=35459,39822,-114130,81825,-122055,-82120,0
C00738=35642,39595,-114632,81591,-122105,-82267,0
C00739=36204,39206,-115497,80959,-122356,-82552,0
C00740=36168,38543,-116954,80794,-122092,-82901,0
C00741=40253,34423,-126058,75646,-123075,-85654,0
C00742=40253,34367,-126057,75664,-123102,-85623,0
C00743=36391,39083,-115658,80780,-122479,-82588,0
C00744=41065,34401,-125997,74869,-123608,-85731,0
C00745=40058,33797,-127300,75688,-122737,-85885,0
C00746=35427,38510,-116905,81501,-121611,-82763,0
C00747=36313,39036,-115761,80838,-122408,-82602,0
C00748=35697,39479,-114778,81537,-122138,-82281,0
C00749=36571,40019,-113600,80902,-122944,-82111,0
C00750=42296,34343,-126143,73624,-124319,-85958,0
C00751=39927,32917,-129217,75565,-122277,-86314,0
C00752=34324,38681,-116514,82563,-120908,-82529,0
C00753=35226,39198,-115388,81884,-121712,-82368,0
C00754=34990,39493,-114737,82185,-121647,-82180,0
C00755=35459,39772,-114129,81841,-122074,-82091,0
C00756=35642,39545,-114631,81606,-122123,-82238,0
C00757=36204,39156,-115495,80974,-122376,-82523,0
C00758=36169,38492,-116953,80810,-122112,-82872,0
C00759=40253,34367,-126057,75664,-123102,-85623,0
C00760=40253,34311,-126054,75681,-123129,-85592,0
C00761=36392,39033,-115656,80796,-122499,-82559,0
C00762=41065,34345,-125995,74888,-123634,-85701,0
C00763=40058,33740,-127298,75706,-122763,-85854,0
C00764=35428,38459,-116902,81516,-121630,-82734,0
C00765=36314,38985,-115759,80854,-122428,-82573,0
C00766=35697,39429,-114776,81552,-122156,-82252,0
C00767=36571,39970,-113599,80918,-122963,-82083,0
C00768=42296,34287,-126141,73643,-124347,-85928,0
C00769=39928,32859,-129214,75582,-122305,-86282,0
C00770=34324,38630,-116512,82578,-120927,-82500,0
C00771=35227,39148,-115386,81900,-121730,-82340,0
C00772=34991,39443,-114736,82201,-121666,-82151,0
C00773=35459,39723,-114127,81856,-122092,-82063,0
C00774=35643,39495,-114629,81622,-122143,-82209,0
C00775=36205,39106,-115494,80990,-122395,-82494,0
C00776=36169,38442,-116952,80826,-122132,-82843,0
C00777=40253,34311,-126054,75681,-123129,-85592,0
C00778=40254,34256,-126053,75699,-123155,-85561,0
C00779=36392,38983,-115654,80812,-122518,-82530,0
C00780=41066,34289,-125992,74906,-123662,-85670,0
C00781=40059,33684,-127297,75723,-122791,-85823,0
C00782=35428,38408,-116901,81532,-121650,-82705,0
C00783=36314,38935,-115758,80870,-122448,-82545,0
C00784=35697,39379,-114775,81568,-122176,-82224,0
C00785=36572,39921,-113597,80934,-122983,-82055,0
C00786=42297,34231,-126139,73662,-124375,-85897,0
C00787=39928,32802,-129213,75600,-122332,-86250,0
C00788=34324,38579,-116511,82593,-120945,-82471,0
C00789=35227,39098,-115384,81915,-121750,-82311,0
C00790=34991,39393,-114734,82216,-121685,-82122,0
C00791=35460,39673,-114125,81872,-122112,-82035,0
C00792=35643,39446,-114627,81637,-122161,-82181,0
C00793=36205,39055,-115491,81006,-122415,-82465,0
C00794=36169,38391,-116950,80841,-122152,-82814,0
C00795=40254,34256,-126053,75699,-123155,-85561,0
C00796=40254,34200,-126051,75717,-123181,-85530,0
C00797=36392,38933,-115652,80828,-122539,-82501,0
C00798=41066,34233,-125991,74924,-123689,-85639,0
C00799=40059,33627,-127294,75741,-122817,-85791,0
C00800=35428,38357,-116899,81547,-121669,-82676,0
C00801=36314,38885,-115756,80886,-122468,-82516,0
C00802=35698,39329,-114773,81584,-122195,-82195,0
C00803=36572,39871,-113595,80950,-123002,-82026,0
C00804=42297,34175,-126137,73680,-124404,-85866,0
C00805=39928,32744,-129211,75617,-122360,-86218,0
C00806=34325,38529,-116508,82607,-120964,-82441,0
C00807=35227,39048,-115382,81931,-121768,-82282,0
C00808=34991,39343,-114732,82231,-121704,-82094,0
C00809=35460,39623,-114123,81887,-122130,-82006,0
C00810=35643,39396,-114626,81653,-122181,-82152,0
C00811=36205,39005,-115490,81022,-122434,-82437,0
C00812=36170,38340,-116947,80857,-122172,-82785,0
C00813=40254,34200,-126051,75717,-123181,-85530,0
C00814=40255,34144,-126049,75735,-123208,-85499,0
C00815=36393,38882,-115650,80844,-122559,-82472,0
C00816=41067,34178,-125989,74942,-123717,-85608,0
C00817=40060,33571,-127292,75759,-122844,-85760,0
C00818=35429,38307,-116897,81563,-121689,-82646,0
C00819=36315,38835,-115753,80902,-122487,-82487,0
C00820=35698,39279,-114771,81599,-122214,-82166,0
C00821=36572,39822,-113593,80967,-123022,-81998,0
C00822=42298,34119,-126135,73699,-124433,-85835,0
C00823=39929,32686,-129209,75635,-122387,-86186,0
C00824=34325,38478,-116506,82622,-120982,-82412,0
C00825=35228,38998,-115381,81946,-121788,-82253,0
C00826=34992,39293,-114730,82246,-121722,-82065,0
C00827=35461,39574,-114121,81903,-122148,-81978,0
C00828=35644,39346,-114624,81669,-122199,-82123,0
C00829=36206,38955,-115488,81038,-122455,-82408,0
C00830=36170,38289,-116946,80873,-122192,-82755,0
C00831=40255,34144,-126049,75735,-123208,-85499,0
C00832=40255,34088,-126047,75753,-123234,-85467,0
C00833=36393,38832,-115649,80861,-122578,-82443,0
C00834=41067,34122,-125987,74960,-123743,-85577,0
C00835=40060,33514,-127291,75776,-122871,-85728,0
C00836=35429,38256,-116896,81578,-121707,-82617,0
C00837=36315,38784,-115752,80918,-122507,-82458,0
C00838=35698,39230,-114769,81615,-122233,-82138,0
C00839=36572,39773,-113591,80983,-123040,-81970,0
C00840=42298,34064,-126134,73718,-124460,-85805,0
C00841=39929,32629,-129206,75653,-122415,-86154,0
C00842=34325,38428,-116505,82637,-121000,-82383,0
C00843=35228,38948,-115379,81962,-121806,-82224,0
C00844=34992,39244,-114728,82262,-121740,-82036,0
C00845=35461,39525,-114120,81919,-122167,-81949,0
C00846=35644,39296,-114622,81685,-122218,-82095,0
C00847=36206,38905,-115486,81054,-122475,-82379,0
C00848=36170,38238,-116944,80889,-122213,-82726,0
C00849=40255,34088,-126047,75753,-123234,-85467,0
C00850=40255,34033,-126045,75771,-123261,-85437,0
C00851=36393,38782,-115646,80877,-122598,-82415,0
C00852=41067,34067,-125984,74979,-123771,-85546,0
C00853=40061,33458,-127289,75794,-122898,-85697,0
C00854=35429,38205,-116893,81594,-121727,-82588,0
C00855=36315,38734,-115750,80934,-122526,-82429,0
C00856=35699,39180,-114767,81631,-122252,-82109,0
C00857=36573,39724,-113589,80999,-123060,-81941,0
C00858=42298,34008,-126131,73737,-124489,-85774,0
C00859=39930,32571,-129205,75670,-122443,-86121,0
C00860=34326,38377,-116503,82652,-121019,-82354,0
C00861=35228,38898,-115376,81977,-121824,-82195,0
C00862=34992,39194,-114726,82277,-121759,-82007,0
C00863=35461,39475,-114117,81934,-122186,-81920,0
C00864=35644,39247,-114620,81700,-122237,-82066,0
C00865=36206,38855,-115484,81070,-122494,-82350,0
C00866=36171,38188,-116942,80905,-122232,-82697,0
C00867=40255,34033,-126045,75771,-123261,-85437,0
C00868=40256,33977,-126043,75789,-123288,-85405,0
C00869=36394,38732,-115644,80893,-122618,-82386,0
C00870=41068,34011,-125982,74997,-123799,-85515,0
C00871=40061,33401,-127286,75812,-122925,-85665,0
C00872=35430,38154,-116891,81609,-121746,-82559,0
C00873=36316,38684,-115748,80950,-122547,-82400,0
C00874=35699,39130,-114765,81647,-122271,-82080,0
C00875=36573,39675,-113587,81015,-123079,-81913,0
C00876=42299,33952,-126129,73756,-124518,-85743,0
C00877=39930,32513,-129203,75688,-122470,-86090,0
C00878=34326,38327,-116500,82667,-121037,-82325,0
C00879=35229,38848,-115374,81993,-121844,-82166,0
C00880=34993,39144,-114724,82293,-121777,-81979,0
C00881=35461,39426,-114115,81950,-122205,-81892,0
C00882=35645,39197,-114617,81716,-122256,-82038,0
C00883=36207,38805,-115482,81086,-122514,-82321,0
C00884=36171,38137,-116939,80921,-122252,-82668,0
C00885=40256,33977,-126043,75789,-123288,-85405,0
C00886=40256,33922,-126041,75807,-123315,-85374,0
C00887=36394,38682,-115642,80909,-122638,-82357,0
C00888=41068,33956,-125980,75015,-123826,-85484,0
C00889=40061,33345,-127284,75830,-122952,-85633,0
C00890=35430,38104,-116889,81625,-121766,-82530,0
C00891=36316,38634,-115745,80966,-122567,-82371,0
C00892=35699,39081,-114762,81663,-122290,-82051,0
C00893=36573,39626,-113585,81032,-123099,-81884,0
C00894=42299,33897,-126127,73775,-124547,-85712,0
C00895=39930,32456,-129200,75706,-122498,-86058,0
C00896=34326,38276,-116498,82682,-121055,-82296,0
C00897=35229,38798,-115372,82008,-121862,-82137,0
C00898=34993,39095,-114722,82308,-121796,-81950,0
C00899=35462,39376,-114113,81966,-122223,-81863,0
C00900=35645,39148,-114615,81732,-122275,-82009,0
C00901=36207,38755,-115480,81102,-122533,-82292,0
C00902=36171,38086,-116937,80937,-122272,-82639,0
C00903=40256,33922,-126041,75807,-123315,-85374,0
C00904=40257,33866,-126038,75825,-123341,-85343,0
C00905=36394,38632,-115640,80925,-122657,-82328,0
C00906=41069,33900,-125977,75034,-123853,-85453,0
C00907=40062,33289,-127280,75848,-122979,-85602,0
C00908=35430,38053,-116886,81641,-121785,-82500,0
C00909=36316,38584,-115743,80982,-122586,-82342,0
C00910=35700,39031,-114760,81679,-122309,-82022,0
C00911=36574,39576,-113583,81048,-123118,-81855,0
C00912=42300,33841,-126124,73794,-124574,-85681,0
C00913=39931,32398,-129197,75724,-122525,-86025,0
C00914=34327,38226,-116496,82697,-121074,-82266,0
C00915=35229,38748,-115369,82024,-121882,-82108,0
C00916=34993,39045,-114719,82324,-121814,-81921,0
C00917=35462,39327,-114111,81981,-122241,-81834,0
C00918=35645,39098,-114613,81748,-122294,-81980,0
C00919=36207,38705,-115477,81119,-122553,-82263,0
C00920=36172,38036,-116935,80953,-122292,-82610,0
C00921=40257,33866,-126038,75825,-123341,-85343,0
C00922=40257,33811,-126035,75843,-123368,-85312,0
C00923=36395,38582,-115637,80942,-122677,-82299,0
C00924=41069,33845,-125975,75052,-123880,-85422,0
C00925=40062,33233,-127278,75866,-123006,-85571,0
C00926=35431,38003,-116884,81656,-121805,-82471,0
C00927=36317,38534,-115741,80999,-122606,-82313,0
C00928=35700,38981,-114758,81695,-122329,-81993,0
C00929=36574,39527,-113580,81065,-123138,-81827,0
C00930=42300,33786,-126121,73813,-124603,-85650,0
C00931=39931,32341,-129195,75742,-122553,-85993,0
C00932=34327,38175,-116493,82713,-121092,-82237,0
C00933=35230,38698,-115367,82039,-121900,-82079,0
C00934=34994,38996,-114717,82339,-121832,-81892,0
C00935=35462,39278,-114108,81997,-122261,-81805,0
C00936=35646,39049,-114610,81764,-122313,-81951,0
C00937=36208,38655,-115475,81135,-122572,-82234,0
C00938=36172,37985,-116932,80970,-122313,-82580,0
C00939=40257,33811,-126035,75843,-123368,-85312,0
C00940=40257,33755,-126032,75861,-123394,-85281,0
C00941=36395,38532,-115635,80958,-122698,-82270,0
C00942=41069,33789,-125973,75071,-123908,-85390,0
C00943=40063,33176,-127276,75884,-123032,-85539,0
C00944=35431,37952,-116882,81672,-121824,-82441,0
C00945=36317,38484,-115738,81015,-122626,-82284,0
C00946=35700,38932,-114755,81710,-122347,-81965,0
C00947=36575,39478,-113578,81081,-123157,-81798,0
C00948=42301,33730,-126119,73832,-124632,-85619,0
C00949=39932,32284,-129193,75759,-122580,-85961,0
C00950=34327,38125,-116491,82728,-121111,-82208,0
C00951=35230,38649,-115365,82055,-121920,-82050,0
C00952=34994,38946,-114714,82355,-121851,-81863,0
C00953=35463,39229,-114106,82013,-122279,-81777,0
C00954=35646,38999,-114608,81779,-122332,-81922,0
C00955=36208,38606,-115472,81151,-122592,-82205,0
C00956=36172,37935,-116930,80986,-122332,-82550,0
C00957=40257,33755,-126032,75861,-123394,-85281,0
C00958=40258,33700,-126030,75879,-123420,-85249,0
C00959=36395,38482,-115631,80974,-122717,-82241,0
C00960=41070,33734,-125969,75089,-123935,-85360,0
C00961=40063,33120,-127274,75902,-123060,-85507,0
C00962=35431,37902,-116878,81688,-121844,-82412,0
C00963=36317,38434,-115735,81031,-122646,-82255,0
C00964=35701,38882,-114752,81726,-122367,-81936,0
C00965=36575,39430,-113575,81097,-123176,-81769,0
C00966=42301,33675,-126116,73851,-124660,-85588,0
C00967=39932,32226,-129189,75778,-122608,-85929,0
C00968=34328,38075,-116488,82743,-121130,-82179,0
C00969=35230,38599,-115363,82071,-121938,-82021,0
C00970=34994,38897,-114712,82370,-121869,-81834,0
C00971=35463,39179,-114103,82029,-122298,-81748,0
C00972=35646,38950,-114605,81795,-122351,-81893,0
C00973=36208,38556,-115469,81167,-122611,-82176,0
C00974=36173,37884,-116928,81002,-122353,-82521,0
C00975=40258,33700,-126030,75879,-123420,-85249,0
C00976=40258,33645,-126027,75897,-123448,-85218,0
C00977=36396,38432,-115629,80991,-122737,-82212,0
C00978=41070,33679,-125967,75108,-123962,-85328,0
C00979=40063,33064,-127270,75920,-123086,-85476,0
C00980=35432,37851,-116876,81704,-121863,-82383,0
C00981=36318,38384,-115733,81048,-122665,-82226,0
C00982=35701,38833,-114750,81742,-122385,-81907,0
C00983=36575,39381,-113573,81114,-123195,-81741,0
C00984=42301,33620,-126113,73870,-124688,-85557,0
C00985=39933,32169,-129187,75795,-122636,-85896,0
C00986=34328,38025,-116485,82758,-121149,-82149,0
C00987=35231,38549,-115359,82086,-121956,-81992,0
C00988=34995,38847,-114709,82386,-121889,-81805,0
C00989=35463,39130,-114101,82045,-122316,-81720,0
C00990=35647,38900,-114603,81811,-122370,-81865,0
C00991=36209,38506,-115467,81183,-122631,-82147,0
C00992=36173,37834,-116924,81018,-122372,-82492,0
C00993=40258,33645,-126027,75897,-123448,-85218,0
C00994=40259,33589,-126024,75915,-123474,-85187,0
C00995=36396,38383,-115627,81007,-122756,-82183,0
C00996=41071,33623,-125965,75126,-123989,-85297,0
C00997=40064,33008,-127268,75938,-123114,-85444,0
C00998=35432,37801,-116874,81720,-121883,-82353,0
C00999=36318,38334,-115730,81064,-122685,-82197,0
C01000=35701,38784,-114747,81758,-122405,-81878,0
C01001=36576,39332,-113570,81130,-123215,-81713,0
C01002=42302,33564,-126111,73889,-124717,-85526,0
C01003=39933,32112,-129183,75813,-122663,-85864,0
C01004=34328,37974,-116483,82773,-121167,-82119,0
C01005=35231,38500,-115357,82102,-121976,-81963,0
C01006=34995,38798,-114706,82401,-121907,-81776,0
C01007=35464,39081,-114098,82061,-122336,-81691,0
C01008=35647,38851,-114600,81827,-122389,-81836,0
C01009=36209,38456,-115464,81200,-122651,-82118,0
C01010=36173,37783,-116922,81034,-122392,-82463,0
C01011=40259,33589,-126024,75915,-123474,-85187,0
C01012=40259,33534,-126021,75934,-123501,-85155,0
C01013=36396,38333,-115623,81023,-122777,-82153,0
C01014=41071,33568,-125961,75145,-124017,-85266,0
C01015=40064,32952,-127264,75956,-123140,-85412,0
C01016=35432,37751,-116870,81736,-121902,-82324,0
C01017=36318,38285,-115727,81080,-122705,-82168,0
C01018=35702,38734,-114744,81774,-122423,-81849,0
C01019=36576,39283,-113567,81147,-123234,-81684,0
C01020=42302,33509,-126107,73908,-124745,-85495,0
C01021=39933,32054,-129181,75832,-122691,-85832,0
C01022=34329,37924,-116480,82788,-121185,-82090,0
C01023=35231,38450,-115353,82118,-121994,-81934,0
C01024=34995,38748,-114704,82417,-121925,-81747,0
C01025=35464,39032,-114095,82076,-122354,-81662,0
C01026=35647,38802,-114597,81843,-122408,-81807,0
C01027=36209,38407,-115461,81216,-122670,-82089,0
C01028=36174,37733,-116920,81051,-122413,-82433,0
C01029=40259,33534,-126021,75934,-123501,-85155,0
C01030=40259,33479,-126019,75952,-123527,-85124,0
C01031=36397,38283,-115621,81040,-122796,-82124,0
C01032=41072,33513,-125958,75164,-124044,-85234,0
C01033=40065,32896,-127261,75974,-123168,-85380,0
C01034=35433,37700,-116868,81751,-121922,-82294,0
C01035=36319,38235,-115725,81097,-122725,-82138,0
C01036=35702,38685,-114741,81790,-122443,-81820,0
C01037=36576,39234,-113564,81163,-123254,-81655,0
C01038=42303,33454,-126105,73928,-124774,-85463,0
C01039=39934,31997,-129178,75850,-122718,-85799,0
C01040=34329,37874,-116477,82804,-121204,-82061,0
C01041=35232,38400,-115351,82134,-122014,-81905,0
C01042=34996,38699,-114701,82433,-121944,-81718,0
C01043=35464,38983,-114092,82092,-122372,-81632,0
C01044=35648,38753,-114594,81859,-122426,-81778,0
C01045=36210,38357,-115458,81232,-122691,-82060,0
C01046=36174,37683,-116916,81067,-122432,-82404,0
C01047=40259,33479,-126019,75952,-123527,-85124,0
C01048=40260,33424,-126015,75970,-123554,-85093,0
C01049=36397,38233,-115618,81056,-122816,-82095,0
C01050=41072,33458,-125955,75183,-124071,-85203,0
C01051=40065,32840,-127259,75993,-123194,-85349,0
C01052=35433,37650,-116865,81767,-121940,-82265,0
C01053=36319,38185,-115721,81113,-122745,-82109,0
C01054=35702,38636,-114738,81807,-122461,-81791,0
C01055=36576,39185,-113561,81180,-123273,-81626,0
C01056=42303,33398,-126101,73947,-124802,-85432,0
C01057=39934,31940,-129174,75868,-122746,-85767,0
C01058=34329,37824,-116474,82819,-121222,-82031,0
C01059=35232,38351,-115348,82150,-122032,-81876,0
C01060=34996,38650,-114698,82448,-121962,-81689,0
C01061=35465,38934,-114089,82108,-122391,-81604,0
C01062=35648,38703,-114591,81875,-122446,-81749,0
C01063=36210,38307,-115456,81249,-122710,-82031,0
C01064=36174,37632,-116913,81083,-122453,-82374,0
C01065=40260,33424,-126015,75970,-123554,-85093,0
C01066=40260,33369,-126012,75989,-123580,-85061,0
C01067=36397,38184,-115614,81073,-122836,-82065,0
C01068=41072,33403,-125952,75201,-124098,-85172,0
C01069=40065,32784,-127255,76011,-123222,-85317,0
C01070=35433,37600,-116861,81783,-121960,-82235,0
C01071=36319,38136,-115718,81130,-122764,-82080,0
C01072=35703,38586,-114735,81823,-122480,-81762,0
C01073=36577,39137,-113558,81197,-123293,-81598,0
C01074=42303,33343,-126098,73966,-124830,-85401,0
C01075=39935,31883,-129171,75886,-122773,-85734,0
C01076=34330,37774,-116470,82834,-121241,-82002,0
C01077=35232,38301,-115345,82166,-122051,-81847,0
C01078=34996,38601,-114695,82464,-121981,-81660,0
C01079=35465,38885,-114086,82124,-122410,-81575,0
C01080=35648,38654,-114588,81892,-122464,-81720,0
C01081=36210,38258,-115452,81265,-122730,-82002,0
C01082=36175,37582,-116910,81100,-122472,-82344,0
C01083=40260,33369,-126012,75989,-123580,-85061,0
C01084=40261,33314,-126008,76007,-123607,-85029,0
C01085=36398,38134,-115612,81089,-122856,-82036,0
C01086=41073,33348,-125949,75220,-124126,-85140,0
C01087=40066,32729,-127252,76029,-123248,-85285,0
C01088=35434,37550,-116859,81799,-121979,-82206,0
C01089=36320,38086,-115715,81146,-122784,-82050,0
C01090=35703,38537,-114732,81839,-122500,-81733,0
C01091=36577,39088,-113555,81213,-123311,-81569,0
C01092=42304,33288,-126095,73986,-124859,-85369,0
C01093=39935,31826,-129169,75904,-122801,-85702,0
C01094=34330,37724,-116468,82850,-121259,-81972,0
C01095=35233,38252,-115342,82181,-122070,-81818,0
C01096=34997,38552,-114692,82480,-121999,-81631,0
C01097=35465,38836,-114083,82140,-122429,-81546,0
C01098=35649,38605,-114585,81908,-122484,-81691,0
C01099=36211,38208,-115449,81282,-122749,-81973,0
C01100=36175,37532,-116907,81116,-122493,-82315,0
C01101=40261,33314,-126008,76007,-123607,-85029,0
C01102=40261,33259,-126005,76026,-123634,-84998,0
C01103=36398,38085,-115608,81106,-122876,-82007,0
C01104=41073,33293,-125945,75239,-124154,-85109,0
C01105=40066,32673,-127248,76048,-123275,-85253,0
C01106=35434,37499,-116855,81815,-121999,-82176,0
C01107=36320,38036,-115712,81163,-122805,-82021,0
C01108=35703,38488,-114729,81855,-122518,-81704,0
C01109=36577,39039,-113552,81230,-123331,-81540,0
C01110=42304,33233,-126091,74005,-124888,-85339,0
C01111=39935,31769,-129165,75923,-122829,-85669,0
C01112=34330,37674,-116465,82865,-121277,-81943,0
C01113=35233,38202,-115338,82197,-122089,-81788,0
C01114=34997,38502,-114688,82496,-122017,-81602,0
C01115=35466,38787,-114080,82157,-122447,-81517,0
C01116=35649,38556,-114582,81924,-122502,-81662,0
C01117=36211,38159,-115446,81298,-122769,-81943,0
C01118=36175,37482,-116904,81133,-122513,-82286,0
C01119=40261,33259,-126005,76026,-123634,-84998,0
C01120=40262,33204,-126001,76044,-123661,-84967,0
C01121=36398,38035,-115605,81123,-122895,-81978,0
C01122=41074,33238,-125942,75258,-124180,-85078,0
C01123=40067,32617,-127245,76066,-123302,-85221,0
C01124=35434,37449,-116852,81831,-122018,-82147,0
C01125=36320,37987,-115708,81179,-122824,-81992,0
C01126=35704,38439,-114726,81871,-122538,-81675,0
C01127=36578,38991,-113548,81247,-123350,-81511,0
C01128=42305,33178,-126088,74025,-124916,-85307,0
C01129=39936,31712,-129160,75941,-122856,-85637,0
C01130=34331,37624,-116461,82881,-121296,-81913,0
C01131=35233,38153,-115335,82213,-122108,-81759,0
C01132=34997,38453,-114685,82512,-122036,-81573,0
C01133=35466,38739,-114076,82173,-122466,-81488,0
C01134=35649,38507,-114579,81940,-122522,-81632,0
C01135=36211,38109,-115443,81315,-122788,-81914,0
C01136=36176,37432,-116900,81149,-122532,-82256,0
C01137=40262,33204,-126001,76044,-123661,-84967,0
C01138=40262,33149,-125998,76063,-123687,-84935,0
C01139=36399,37986,-115602,81139,-122915,-81949,0
C01140=41074,33183,-125938,75277,-124208,-85046,0
C01141=40067,32561,-127241,76084,-123329,-85189,0
C01142=35434,37399,-116848,81847,-122038,-82117,0
C01143=36321,37937,-115705,81196,-122844,-81963,0
C01144=35704,38390,-114722,81888,-122556,-81646,0
C01145=36578,38942,-113545,81264,-123370,-81482,0
C01146=42305,33123,-126084,74044,-124944,-85276,0
C01147=39936,31655,-129157,75959,-122885,-85604,0
C01148=34331,37574,-116458,82896,-121314,-81884,0
C01149=35234,38104,-115332,82229,-122127,-81729,0
C01150=34997,38404,-114682,82527,-122054,-81544,0
C01151=35466,38690,-114073,82189,-122485,-81459,0
C01152=35650,38458,-114575,81956,-122540,-81603,0
C01153=36212,38060,-115440,81331,-122808,-81884,0
C01154=36176,37382,-116897,81166,-122553,-82227,0
C01155=40262,33149,-125998,76063,-123687,-84935,0
C01156=40262,33094,-125995,76081,-123713,-84903,0
C01157=36399,37936,-115598,81156,-122936,-81919,0
C01158=41074,33128,-125935,75296,-124235,-85015,0
C01159=40067,32506,-127238,76103,-123356,-85157,0
C01160=35435,37349,-116845,81864,-122058,-82087,0
C01161=36321,37888,-115702,81212,-122863,-81933,0
//INST
///DATE 2025/02/20 16:20
///COMM Generated using RoboDK
///ATTR SC,RW
///GROUP1 RB1
NOP
MOVL C00000 V=30.0 PL=1
MOVL C00001 V=130.0 PL=1
MOVL C00002 V=130.0 PL=1
MOVL C00003 V=20.0 PL=1
MOVL C00004 V=130.0 PL=1
MOVL C00005 V=130.0 PL=1
MOVL C00006 V=60.0 PL=1
MOVL C00007 V=60.0 PL=1
MOVL C00008 V=60.0 PL=1
MOVL C00009 V=60.0 PL=1
MOVL C00010 V=130.0 PL=1
MOVL C00011 V=30.0 PL=1
MOVL C00012 V=30.0 PL=1
MOVL C00013 V=30.0 PL=1
MOVL C00014 V=30.0 PL=1
MOVL C00015 V=30.0 PL=1
MOVL C00016 V=30.0 PL=1
MOVL C00017 V=30.0 PL=1
MOVL C00018 V=30.0 PL=1
MOVL C00019 V=130.0 PL=1
MOVL C00020 V=130.0 PL=1
MOVL C00021 V=20.0 PL=1
MOVL C00022 V=130.0 PL=1
MOVL C00023 V=130.0 PL=1
MOVL C00024 V=60.0 PL=1
MOVL C00025 V=60.0 PL=1
MOVL C00026 V=60.0 PL=1
MOVL C00027 V=60.0 PL=1
MOVL C00028 V=130.0 PL=1
MOVL C00029 V=30.0 PL=1
MOVL C00030 V=30.0 PL=1
MOVL C00031 V=30.0 PL=1
MOVL C00032 V=30.0 PL=1
MOVL C00033 V=30.0 PL=1
MOVL C00034 V=30.0 PL=1
MOVL C00035 V=30.0 PL=1
MOVL C00036 V=30.0 PL=1
MOVL C00037 V=130.0 PL=1
MOVL C00038 V=130.0 PL=1
MOVL C00039 V=20.0 PL=1
MOVL C00040 V=130.0 PL=1
MOVL C00041 V=130.0 PL=1
MOVL C00042 V=60.0 PL=1
MOVL C00043 V=60.0 PL=1
MOVL C00044 V=60.0 PL=1
MOVL C00045 V=60.0 PL=1
MOVL C00046 V=130.0 PL=1
MOVL C00047 V=30.0 PL=1
MOVL C00048 V=30.0 PL=1
MOVL C00049 V=30.0 PL=1
MOVL C00050 V=30.0 PL=1
MOVL C00051 V=30.0 PL=1
MOVL C00052 V=30.0 PL=1
MOVL C00053 V=30.0 PL=1
MOVL C00054 V=30.0 PL=1
MOVL C00055 V=130.0 PL=1
MOVL C00056 V=130.0 PL=1
MOVL C00057 V=20.0 PL=1
MOVL C00058 V=130.0 PL=1
MOVL C00059 V=130.0 PL=1
MOVL C00060 V=60.0 PL=1
MOVL C00061 V=60.0 PL=1
MOVL C00062 V=60.0 PL=1
MOVL C00063 V=60.0 PL=1
MOVL C00064 V=130.0 PL=1
MOVL C00065 V=30.0 PL=1
MOVL C00066 V=30.0 PL=1
MOVL C00067 V=30.0 PL=1
MOVL C00068 V=30.0 PL=1
MOVL C00069 V=30.0 PL=1
MOVL C00070 V=30.0 PL=1
MOVL C00071 V=30.0 PL=1
MOVL C00072 V=30.0 PL=1
MOVL C00073 V=130.0 PL=1
MOVL C00074 V=130.0 PL=1
MOVL C00075 V=20.0 PL=1
MOVL C00076 V=130.0 PL=1
MOVL C00077 V=130.0 PL=1
MOVL C00078 V=60.0 PL=1
MOVL C00079 V=60.0 PL=1
MOVL C00080 V=60.0 PL=1
MOVL C00081 V=60.0 PL=1
MOVL C00082 V=130.0 PL=1
MOVL C00083 V=30.0 PL=1
MOVL C00084 V=30.0 PL=1
MOVL C00085 V=30.0 PL=1
MOVL C00086 V=30.0 PL=1
MOVL C00087 V=30.0 PL=1
MOVL C00088 V=30.0 PL=1
MOVL C00089 V=30.0 PL=1
MOVL C00090 V=30.0 PL=1
MOVL C00091 V=130.0 PL=1
MOVL C00092 V=130.0 PL=1
MOVL C00093 V=20.0 PL=1
MOVL C00094 V=130.0 PL=1
MOVL C00095 V=130.0 PL=1
MOVL C00096 V=60.0 PL=1
MOVL C00097 V=60.0 PL=1
MOVL C00098 V=60.0 PL=1
MOVL C00099 V=60.0 PL=1
MOVL C00100 V=130.0 PL=1
MOVL C00101 V=30.0 PL=1
MOVL C00102 V=30.0 PL=1
MOVL C00103 V=30.0 PL=1
MOVL C00104 V=30.0 PL=1
MOVL C00105 V=30.0 PL=1
MOVL C00106 V=30.0 PL=1
MOVL C00107 V=30.0 PL=1
MOVL C00108 V=30.0 PL=1
MOVL C00109 V=130.0 PL=1
MOVL C00110 V=130.0 PL=1
MOVL C00111 V=20.0 PL=1
MOVL C00112 V=130.0 PL=1
MOVL C00113 V=130.0 PL=1
MOVL C00114 V=60.0 PL=1
MOVL C00115 V=60.0 PL=1
MOVL C00116 V=60.0 PL=1
MOVL C00117 V=60.0 PL=1
MOVL C00118 V=130.0 PL=1
MOVL C00119 V=30.0 PL=1
MOVL C00120 V=30.0 PL=1
MOVL C00121 V=30.0 PL=1
MOVL C00122 V=30.0 PL=1
MOVL C00123 V=30.0 PL=1
MOVL C00124 V=30.0 PL=1
MOVL C00125 V=30.0 PL=1
MOVL C00126 V=30.0 PL=1
MOVL C00127 V=130.0 PL=1
MOVL C00128 V=130.0 PL=1
MOVL C00129 V=20.0 PL=1
MOVL C00130 V=130.0 PL=1
MOVL C00131 V=130.0 PL=1
MOVL C00132 V=60.0 PL=1
MOVL C00133 V=60.0 PL=1
MOVL C00134 V=60.0 PL=1
MOVL C00135 V=60.0 PL=1
MOVL C00136 V=130.0 PL=1
MOVL C00137 V=30.0 PL=1
MOVL C00138 V=30.0 PL=1
MOVL C00139 V=30.0 PL=1
MOVL C00140 V=30.0 PL=1
MOVL C00141 V=30.0 PL=1
MOVL C00142 V=30.0 PL=1
MOVL C00143 V=30.0 PL=1
MOVL C00144 V=30.0 PL=1
MOVL C00145 V=130.0 PL=1
MOVL C00146 V=130.0 PL=1
MOVL C00147 V=20.0 PL=1
MOVL C00148 V=130.0 PL=1
MOVL C00149 V=130.0 PL=1
MOVL C00150 V=60.0 PL=1
MOVL C00151 V=60.0 PL=1
MOVL C00152 V=60.0 PL=1
MOVL C00153 V=60.0 PL=1
MOVL C00154 V=130.0 PL=1
MOVL C00155 V=30.0 PL=1
MOVL C00156 V=30.0 PL=1
MOVL C00157 V=30.0 PL=1
MOVL C00158 V=30.0 PL=1
MOVL C00159 V=30.0 PL=1
MOVL C00160 V=30.0 PL=1
MOVL C00161 V=30.0 PL=1
MOVL C00162 V=30.0 PL=1
MOVL C00163 V=130.0 PL=1
MOVL C00164 V=130.0 PL=1
MOVL C00165 V=20.0 PL=1
MOVL C00166 V=130.0 PL=1
MOVL C00167 V=130.0 PL=1
MOVL C00168 V=60.0 PL=1
MOVL C00169 V=60.0 PL=1
MOVL C00170 V=60.0 PL=1
MOVL C00171 V=60.0 PL=1
MOVL C00172 V=130.0 PL=1
MOVL C00173 V=30.0 PL=1
MOVL C00174 V=30.0 PL=1
MOVL C00175 V=30.0 PL=1
MOVL C00176 V=30.0 PL=1
MOVL C00177 V=30.0 PL=1
MOVL C00178 V=30.0 PL=1
MOVL C00179 V=30.0 PL=1
MOVL C00180 V=30.0 PL=1
MOVL C00181 V=130.0 PL=1
MOVL C00182 V=130.0 PL=1
MOVL C00183 V=20.0 PL=1
MOVL C00184 V=130.0 PL=1
MOVL C00185 V=130.0 PL=1
MOVL C00186 V=60.0 PL=1
MOVL C00187 V=60.0 PL=1
MOVL C00188 V=60.0 PL=1
MOVL C00189 V=60.0 PL=1
MOVL C00190 V=130.0 PL=1
MOVL C00191 V=30.0 PL=1
MOVL C00192 V=30.0 PL=1
MOVL C00193 V=30.0 PL=1
MOVL C00194 V=30.0 PL=1
MOVL C00195 V=30.0 PL=1
MOVL C00196 V=30.0 PL=1
MOVL C00197 V=30.0 PL=1
MOVL C00198 V=30.0 PL=1
MOVL C00199 V=130.0 PL=1
MOVL C00200 V=130.0 PL=1
MOVL C00201 V=20.0 PL=1
MOVL C00202 V=130.0 PL=1
MOVL C00203 V=130.0 PL=1
MOVL C00204 V=60.0 PL=1
MOVL C00205 V=60.0 PL=1
MOVL C00206 V=60.0 PL=1
MOVL C00207 V=60.0 PL=1
MOVL C00208 V=130.0 PL=1
MOVL C00209 V=30.0 PL=1
MOVL C00210 V=30.0 PL=1
MOVL C00211 V=30.0 PL=1
MOVL C00212 V=30.0 PL=1
MOVL C00213 V=30.0 PL=1
MOVL C00214 V=30.0 PL=1
MOVL C00215 V=30.0 PL=1
MOVL C00216 V=30.0 PL=1
MOVL C00217 V=130.0 PL=1
MOVL C00218 V=130.0 PL=1
MOVL C00219 V=20.0 PL=1
MOVL C00220 V=130.0 PL=1
MOVL C00221 V=130.0 PL=1
MOVL C00222 V=60.0 PL=1
MOVL C00223 V=60.0 PL=1
MOVL C00224 V=60.0 PL=1
MOVL C00225 V=60.0 PL=1
MOVL C00226 V=130.0 PL=1
MOVL C00227 V=30.0 PL=1
MOVL C00228 V=30.0 PL=1
MOVL C00229 V=30.0 PL=1
MOVL C00230 V=30.0 PL=1
MOVL C00231 V=30.0 PL=1
MOVL C00232 V=30.0 PL=1
MOVL C00233 V=30.0 PL=1
MOVL C00234 V=30.0 PL=1
MOVL C00235 V=130.0 PL=1
MOVL C00236 V=130.0 PL=1
MOVL C00237 V=20.0 PL=1
MOVL C00238 V=130.0 PL=1
MOVL C00239 V=130.0 PL=1
MOVL C00240 V=60.0 PL=1
MOVL C00241 V=60.0 PL=1
MOVL C00242 V=60.0 PL=1
MOVL C00243 V=60.0 PL=1
MOVL C00244 V=130.0 PL=1
MOVL C00245 V=30.0 PL=1
MOVL C00246 V=30.0 PL=1
MOVL C00247 V=30.0 PL=1
MOVL C00248 V=30.0 PL=1
MOVL C00249 V=30.0 PL=1
MOVL C00250 V=30.0 PL=1
MOVL C00251 V=30.0 PL=1
MOVL C00252 V=30.0 PL=1
MOVL C00253 V=130.0 PL=1
MOVL C00254 V=130.0 PL=1
MOVL C00255 V=20.0 PL=1
MOVL C00256 V=130.0 PL=1
MOVL C00257 V=130.0 PL=1
MOVL C00258 V=60.0 PL=1
MOVL C00259 V=60.0 PL=1
MOVL C00260 V=60.0 PL=1
MOVL C00261 V=60.0 PL=1
MOVL C00262 V=130.0 PL=1
MOVL C00263 V=30.0 PL=1
MOVL C00264 V=30.0 PL=1
MOVL C00265 V=30.0 PL=1
MOVL C00266 V=30.0 PL=1
MOVL C00267 V=30.0 PL=1
MOVL C00268 V=30.0 PL=1
MOVL C00269 V=30.0 PL=1
MOVL C00270 V=30.0 PL=1
MOVL C00271 V=130.0 PL=1
MOVL C00272 V=130.0 PL=1
MOVL C00273 V=20.0 PL=1
MOVL C00274 V=130.0 PL=1
MOVL C00275 V=130.0 PL=1
MOVL C00276 V=60.0 PL=1
MOVL C00277 V=60.0 PL=1
MOVL C00278 V=60.0 PL=1
MOVL C00279 V=60.0 PL=1
MOVL C00280 V=130.0 PL=1
MOVL C00281 V=30.0 PL=1
MOVL C00282 V=30.0 PL=1
MOVL C00283 V=30.0 PL=1
MOVL C00284 V=30.0 PL=1
MOVL C00285 V=30.0 PL=1
MOVL C00286 V=30.0 PL=1
MOVL C00287 V=30.0 PL=1
MOVL C00288 V=30.0 PL=1
MOVL C00289 V=130.0 PL=1
MOVL C00290 V=130.0 PL=1
MOVL C00291 V=20.0 PL=1
MOVL C00292 V=130.0 PL=1
MOVL C00293 V=130.0 PL=1
MOVL C00294 V=60.0 PL=1
MOVL C00295 V=60.0 PL=1
MOVL C00296 V=60.0 PL=1
MOVL C00297 V=60.0 PL=1
MOVL C00298 V=130.0 PL=1
MOVL C00299 V=30.0 PL=1
MOVL C00300 V=30.0 PL=1
MOVL C00301 V=30.0 PL=1
MOVL C00302 V=30.0 PL=1
MOVL C00303 V=30.0 PL=1
MOVL C00304 V=30.0 PL=1
MOVL C00305 V=30.0 PL=1
MOVL C00306 V=30.0 PL=1
MOVL C00307 V=130.0 PL=1
MOVL C00308 V=130.0 PL=1
MOVL C00309 V=20.0 PL=1
MOVL C00310 V=130.0 PL=1
MOVL C00311 V=130.0 PL=1
MOVL C00312 V=60.0 PL=1
MOVL C00313 V=60.0 PL=1
MOVL C00314 V=60.0 PL=1
MOVL C00315 V=60.0 PL=1
MOVL C00316 V=130.0 PL=1
MOVL C00317 V=30.0 PL=1
MOVL C00318 V=30.0 PL=1
MOVL C00319 V=30.0 PL=1
MOVL C00320 V=30.0 PL=1
MOVL C00321 V=30.0 PL=1
MOVL C00322 V=30.0 PL=1
MOVL C00323 V=30.0 PL=1
MOVL C00324 V=30.0 PL=1
MOVL C00325 V=130.0 PL=1
MOVL C00326 V=130.0 PL=1
MOVL C00327 V=20.0 PL=1
MOVL C00328 V=130.0 PL=1
MOVL C00329 V=130.0 PL=1
MOVL C00330 V=60.0 PL=1
MOVL C00331 V=60.0 PL=1
MOVL C00332 V=60.0 PL=1
MOVL C00333 V=60.0 PL=1
MOVL C00334 V=130.0 PL=1
MOVL C00335 V=30.0 PL=1
MOVL C00336 V=30.0 PL=1
MOVL C00337 V=30.0 PL=1
MOVL C00338 V=30.0 PL=1
MOVL C00339 V=30.0 PL=1
MOVL C00340 V=30.0 PL=1
MOVL C00341 V=30.0 PL=1
MOVL C00342 V=30.0 PL=1
MOVL C00343 V=130.0 PL=1
MOVL C00344 V=130.0 PL=1
MOVL C00345 V=20.0 PL=1
MOVL C00346 V=130.0 PL=1
MOVL C00347 V=130.0 PL=1
MOVL C00348 V=60.0 PL=1
MOVL C00349 V=60.0 PL=1
MOVL C00350 V=60.0 PL=1
MOVL C00351 V=60.0 PL=1
MOVL C00352 V=130.0 PL=1
MOVL C00353 V=30.0 PL=1
MOVL C00354 V=30.0 PL=1
MOVL C00355 V=30.0 PL=1
MOVL C00356 V=30.0 PL=1
MOVL C00357 V=30.0 PL=1
MOVL C00358 V=30.0 PL=1
MOVL C00359 V=30.0 PL=1
MOVL C00360 V=30.0 PL=1
MOVL C00361 V=130.0 PL=1
MOVL C00362 V=130.0 PL=1
MOVL C00363 V=20.0 PL=1
MOVL C00364 V=130.0 PL=1
MOVL C00365 V=130.0 PL=1
MOVL C00366 V=60.0 PL=1
MOVL C00367 V=60.0 PL=1
MOVL C00368 V=60.0 PL=1
MOVL C00369 V=60.0 PL=1
MOVL C00370 V=130.0 PL=1
MOVL C00371 V=30.0 PL=1
MOVL C00372 V=30.0 PL=1
MOVL C00373 V=30.0 PL=1
MOVL C00374 V=30.0 PL=1
MOVL C00375 V=30.0 PL=1
MOVL C00376 V=30.0 PL=1
MOVL C00377 V=30.0 PL=1
MOVL C00378 V=30.0 PL=1
MOVL C00379 V=130.0 PL=1
MOVL C00380 V=130.0 PL=1
MOVL C00381 V=20.0 PL=1
MOVL C00382 V=130.0 PL=1
MOVL C00383 V=130.0 PL=1
MOVL C00384 V=60.0 PL=1
MOVL C00385 V=60.0 PL=1
MOVL C00386 V=60.0 PL=1
MOVL C00387 V=60.0 PL=1
MOVL C00388 V=130.0 PL=1
MOVL C00389 V=30.0 PL=1
MOVL C00390 V=30.0 PL=1
MOVL C00391 V=30.0 PL=1
MOVL C00392 V=30.0 PL=1
MOVL C00393 V=30.0 PL=1
MOVL C00394 V=30.0 PL=1
MOVL C00395 V=30.0 PL=1
MOVL C00396 V=30.0 PL=1
MOVL C00397 V=130.0 PL=1
MOVL C00398 V=130.0 PL=1
MOVL C00399 V=20.0 PL=1
MOVL C00400 V=130.0 PL=1
MOVL C00401 V=130.0 PL=1
MOVL C00402 V=60.0 PL=1
MOVL C00403 V=60.0 PL=1
MOVL C00404 V=60.0 PL=1
MOVL C00405 V=60.0 PL=1
MOVL C00406 V=130.0 PL=1
MOVL C00407 V=30.0 PL=1
MOVL C00408 V=30.0 PL=1
MOVL C00409 V=30.0 PL=1
MOVL C00410 V=30.0 PL=1
MOVL C00411 V=30.0 PL=1
MOVL C00412 V=30.0 PL=1
MOVL C00413 V=30.0 PL=1
MOVL C00414 V=30.0 PL=1
MOVL C00415 V=130.0 PL=1
MOVL C00416 V=130.0 PL=1
MOVL C00417 V=20.0 PL=1
MOVL C00418 V=130.0 PL=1
MOVL C00419 V=130.0 PL=1
MOVL C00420 V=60.0 PL=1
MOVL C00421 V=60.0 PL=1
MOVL C00422 V=60.0 PL=1
MOVL C00423 V=60.0 PL=1
MOVL C00424 V=130.0 PL=1
MOVL C00425 V=30.0 PL=1
MOVL C00426 V=30.0 PL=1
MOVL C00427 V=30.0 PL=1
MOVL C00428 V=30.0 PL=1
MOVL C00429 V=30.0 PL=1
MOVL C00430 V=30.0 PL=1
MOVL C00431 V=30.0 PL=1
MOVL C00432 V=30.0 PL=1
MOVL C00433 V=130.0 PL=1
MOVL C00434 V=130.0 PL=1
MOVL C00435 V=20.0 PL=1
MOVL C00436 V=130.0 PL=1
MOVL C00437 V=130.0 PL=1
MOVL C00438 V=60.0 PL=1
MOVL C00439 V=60.0 PL=1
MOVL C00440 V=60.0 PL=1
MOVL C00441 V=60.0 PL=1
MOVL C00442 V=130.0 PL=1
MOVL C00443 V=30.0 PL=1
MOVL C00444 V=30.0 PL=1
MOVL C00445 V=30.0 PL=1
MOVL C00446 V=30.0 PL=1
MOVL C00447 V=30.0 PL=1
MOVL C00448 V=30.0 PL=1
MOVL C00449 V=30.0 PL=1
MOVL C00450 V=30.0 PL=1
MOVL C00451 V=130.0 PL=1
MOVL C00452 V=130.0 PL=1
MOVL C00453 V=20.0 PL=1
MOVL C00454 V=130.0 PL=1
MOVL C00455 V=130.0 PL=1
MOVL C00456 V=60.0 PL=1
MOVL C00457 V=60.0 PL=1
MOVL C00458 V=60.0 PL=1
MOVL C00459 V=60.0 PL=1
MOVL C00460 V=130.0 PL=1
MOVL C00461 V=30.0 PL=1
MOVL C00462 V=30.0 PL=1
MOVL C00463 V=30.0 PL=1
MOVL C00464 V=30.0 PL=1
MOVL C00465 V=30.0 PL=1
MOVL C00466 V=30.0 PL=1
MOVL C00467 V=30.0 PL=1
MOVL C00468 V=30.0 PL=1
MOVL C00469 V=130.0 PL=1
MOVL C00470 V=130.0 PL=1
MOVL C00471 V=20.0 PL=1
MOVL C00472 V=130.0 PL=1
MOVL C00473 V=130.0 PL=1
MOVL C00474 V=60.0 PL=1
MOVL C00475 V=60.0 PL=1
MOVL C00476 V=60.0 PL=1
MOVL C00477 V=60.0 PL=1
MOVL C00478 V=130.0 PL=1
MOVL C00479 V=30.0 PL=1
MOVL C00480 V=30.0 PL=1
MOVL C00481 V=30.0 PL=1
MOVL C00482 V=30.0 PL=1
MOVL C00483 V=30.0 PL=1
MOVL C00484 V=30.0 PL=1
MOVL C00485 V=30.0 PL=1
MOVL C00486 V=30.0 PL=1
MOVL C00487 V=130.0 PL=1
MOVL C00488 V=130.0 PL=1
MOVL C00489 V=20.0 PL=1
MOVL C00490 V=130.0 PL=1
MOVL C00491 V=130.0 PL=1
MOVL C00492 V=60.0 PL=1
MOVL C00493 V=60.0 PL=1
MOVL C00494 V=60.0 PL=1
MOVL C00495 V=60.0 PL=1
MOVL C00496 V=130.0 PL=1
MOVL C00497 V=30.0 PL=1
MOVL C00498 V=30.0 PL=1
MOVL C00499 V=30.0 PL=1
MOVL C00500 V=30.0 PL=1
MOVL C00501 V=30.0 PL=1
MOVL C00502 V=30.0 PL=1
MOVL C00503 V=30.0 PL=1
MOVL C00504 V=30.0 PL=1
MOVL C00505 V=130.0 PL=1
MOVL C00506 V=130.0 PL=1
MOVL C00507 V=20.0 PL=1
MOVL C00508 V=130.0 PL=1
MOVL C00509 V=130.0 PL=1
MOVL C00510 V=60.0 PL=1
MOVL C00511 V=60.0 PL=1
MOVL C00512 V=60.0 PL=1
MOVL C00513 V=60.0 PL=1
MOVL C00514 V=130.0 PL=1
MOVL C00515 V=30.0 PL=1
MOVL C00516 V=30.0 PL=1
MOVL C00517 V=30.0 PL=1
MOVL C00518 V=30.0 PL=1
MOVL C00519 V=30.0 PL=1
MOVL C00520 V=30.0 PL=1
MOVL C00521 V=30.0 PL=1
MOVL C00522 V=30.0 PL=1
MOVL C00523 V=130.0 PL=1
MOVL C00524 V=130.0 PL=1
MOVL C00525 V=20.0 PL=1
MOVL C00526 V=130.0 PL=1
MOVL C00527 V=130.0 PL=1
MOVL C00528 V=60.0 PL=1
MOVL C00529 V=60.0 PL=1
MOVL C00530 V=60.0 PL=1
MOVL C00531 V=60.0 PL=1
MOVL C00532 V=130.0 PL=1
MOVL C00533 V=30.0 PL=1
MOVL C00534 V=30.0 PL=1
MOVL C00535 V=30.0 PL=1
MOVL C00536 V=30.0 PL=1
MOVL C00537 V=30.0 PL=1
MOVL C00538 V=30.0 PL=1
MOVL C00539 V=30.0 PL=1
MOVL C00540 V=30.0 PL=1
MOVL C00541 V=130.0 PL=1
MOVL C00542 V=130.0 PL=1
MOVL C00543 V=20.0 PL=1
MOVL C00544 V=130.0 PL=1
MOVL C00545 V=130.0 PL=1
MOVL C00546 V=60.0 PL=1
MOVL C00547 V=60.0 PL=1
MOVL C00548 V=60.0 PL=1
MOVL C00549 V=60.0 PL=1
MOVL C00550 V=130.0 PL=1
MOVL C00551 V=30.0 PL=1
MOVL C00552 V=30.0 PL=1
MOVL C00553 V=30.0 PL=1
MOVL C00554 V=30.0 PL=1
MOVL C00555 V=30.0 PL=1
MOVL C00556 V=30.0 PL=1
MOVL C00557 V=30.0 PL=1
MOVL C00558 V=30.0 PL=1
MOVL C00559 V=130.0 PL=1
MOVL C00560 V=130.0 PL=1
MOVL C00561 V=20.0 PL=1
MOVL C00562 V=130.0 PL=1
MOVL C00563 V=130.0 PL=1
MOVL C00564 V=60.0 PL=1
MOVL C00565 V=60.0 PL=1
MOVL C00566 V=60.0 PL=1
MOVL C00567 V=60.0 PL=1
MOVL C00568 V=130.0 PL=1
MOVL C00569 V=30.0 PL=1
MOVL C00570 V=30.0 PL=1
MOVL C00571 V=30.0 PL=1
MOVL C00572 V=30.0 PL=1
MOVL C00573 V=30.0 PL=1
MOVL C00574 V=30.0 PL=1
MOVL C00575 V=30.0 PL=1
MOVL C00576 V=30.0 PL=1
MOVL C00577 V=130.0 PL=1
MOVL C00578 V=130.0 PL=1
MOVL C00579 V=20.0 PL=1
MOVL C00580 V=130.0 PL=1
MOVL C00581 V=130.0 PL=1
MOVL C00582 V=60.0 PL=1
MOVL C00583 V=60.0 PL=1
MOVL C00584 V=60.0 PL=1
MOVL C00585 V=60.0 PL=1
MOVL C00586 V=130.0 PL=1
MOVL C00587 V=30.0 PL=1
MOVL C00588 V=30.0 PL=1
MOVL C00589 V=30.0 PL=1
MOVL C00590 V=30.0 PL=1
MOVL C00591 V=30.0 PL=1
MOVL C00592 V=30.0 PL=1
MOVL C00593 V=30.0 PL=1
MOVL C00594 V=30.0 PL=1
MOVL C00595 V=130.0 PL=1
MOVL C00596 V=130.0 PL=1
MOVL C00597 V=20.0 PL=1
MOVL C00598 V=130.0 PL=1
MOVL C00599 V=130.0 PL=1
MOVL C00600 V=60.0 PL=1
MOVL C00601 V=60.0 PL=1
MOVL C00602 V=60.0 PL=1
MOVL C00603 V=60.0 PL=1
MOVL C00604 V=130.0 PL=1
MOVL C00605 V=30.0 PL=1
MOVL C00606 V=30.0 PL=1
MOVL C00607 V=30.0 PL=1
MOVL C00608 V=30.0 PL=1
MOVL C00609 V=30.0 PL=1
MOVL C00610 V=30.0 PL=1
MOVL C00611 V=30.0 PL=1
MOVL C00612 V=30.0 PL=1
MOVL C00613 V=130.0 PL=1
MOVL C00614 V=130.0 PL=1
MOVL C00615 V=20.0 PL=1
MOVL C00616 V=130.0 PL=1
MOVL C00617 V=130.0 PL=1
MOVL C00618 V=60.0 PL=1
MOVL C00619 V=60.0 PL=1
MOVL C00620 V=60.0 PL=1
MOVL C00621 V=60.0 PL=1
MOVL C00622 V=130.0 PL=1
MOVL C00623 V=30.0 PL=1
MOVL C00624 V=30.0 PL=1
MOVL C00625 V=30.0 PL=1
MOVL C00626 V=30.0 PL=1
MOVL C00627 V=30.0 PL=1
MOVL C00628 V=30.0 PL=1
MOVL C00629 V=30.0 PL=1
MOVL C00630 V=30.0 PL=1
MOVL C00631 V=130.0 PL=1
MOVL C00632 V=130.0 PL=1
MOVL C00633 V=20.0 PL=1
MOVL C00634 V=130.0 PL=1
MOVL C00635 V=130.0 PL=1
MOVL C00636 V=60.0 PL=1
MOVL C00637 V=60.0 PL=1
MOVL C00638 V=60.0 PL=1
MOVL C00639 V=60.0 PL=1
MOVL C00640 V=130.0 PL=1
MOVL C00641 V=30.0 PL=1
MOVL C00642 V=30.0 PL=1
MOVL C00643 V=30.0 PL=1
MOVL C00644 V=30.0 PL=1
MOVL C00645 V=30.0 PL=1
MOVL C00646 V=30.0 PL=1
MOVL C00647 V=30.0 PL=1
MOVL C00648 V=30.0 PL=1
MOVL C00649 V=130.0 PL=1
MOVL C00650 V=130.0 PL=1
MOVL C00651 V=20.0 PL=1
MOVL C00652 V=130.0 PL=1
MOVL C00653 V=130.0 PL=1
MOVL C00654 V=60.0 PL=1
MOVL C00655 V=60.0 PL=1
MOVL C00656 V=60.0 PL=1
MOVL C00657 V=60.0 PL=1
MOVL C00658 V=130.0 PL=1
MOVL C00659 V=30.0 PL=1
MOVL C00660 V=30.0 PL=1
MOVL C00661 V=30.0 PL=1
MOVL C00662 V=30.0 PL=1
MOVL C00663 V=30.0 PL=1
MOVL C00664 V=30.0 PL=1
MOVL C00665 V=30.0 PL=1
MOVL C00666 V=30.0 PL=1
MOVL C00667 V=130.0 PL=1
MOVL C00668 V=130.0 PL=1
MOVL C00669 V=20.0 PL=1
MOVL C00670 V=130.0 PL=1
MOVL C00671 V=130.0 PL=1
MOVL C00672 V=60.0 PL=1
MOVL C00673 V=60.0 PL=1
MOVL C00674 V=60.0 PL=1
MOVL C00675 V=60.0 PL=1
MOVL C00676 V=130.0 PL=1
MOVL C00677 V=30.0 PL=1
MOVL C00678 V=30.0 PL=1
MOVL C00679 V=30.0 PL=1
MOVL C00680 V=30.0 PL=1
MOVL C00681 V=30.0 PL=1
MOVL C00682 V=30.0 PL=1
MOVL C00683 V=30.0 PL=1
MOVL C00684 V=30.0 PL=1
MOVL C00685 V=130.0 PL=1
MOVL C00686 V=130.0 PL=1
MOVL C00687 V=20.0 PL=1
MOVL C00688 V=130.0 PL=1
MOVL C00689 V=130.0 PL=1
MOVL C00690 V=60.0 PL=1
MOVL C00691 V=60.0 PL=1
MOVL C00692 V=60.0 PL=1
MOVL C00693 V=60.0 PL=1
MOVL C00694 V=130.0 PL=1
MOVL C00695 V=30.0 PL=1
MOVL C00696 V=30.0 PL=1
MOVL C00697 V=30.0 PL=1
MOVL C00698 V=30.0 PL=1
MOVL C00699 V=30.0 PL=1
MOVL C00700 V=30.0 PL=1
MOVL C00701 V=30.0 PL=1
MOVL C00702 V=30.0 PL=1
MOVL C00703 V=130.0 PL=1
MOVL C00704 V=130.0 PL=1
MOVL C00705 V=20.0 PL=1
MOVL C00706 V=130.0 PL=1
MOVL C00707 V=130.0 PL=1
MOVL C00708 V=60.0 PL=1
MOVL C00709 V=60.0 PL=1
MOVL C00710 V=60.0 PL=1
MOVL C00711 V=60.0 PL=1
MOVL C00712 V=130.0 PL=1
MOVL C00713 V=30.0 PL=1
MOVL C00714 V=30.0 PL=1
MOVL C00715 V=30.0 PL=1
MOVL C00716 V=30.0 PL=1
MOVL C00717 V=30.0 PL=1
MOVL C00718 V=30.0 PL=1
MOVL C00719 V=30.0 PL=1
MOVL C00720 V=30.0 PL=1
MOVL C00721 V=130.0 PL=1
MOVL C00722 V=130.0 PL=1
MOVL C00723 V=20.0 PL=1
MOVL C00724 V=130.0 PL=1
MOVL C00725 V=130.0 PL=1
MOVL C00726 V=60.0 PL=1
MOVL C00727 V=60.0 PL=1
MOVL C00728 V=60.0 PL=1
MOVL C00729 V=60.0 PL=1
MOVL C00730 V=130.0 PL=1
MOVL C00731 V=30.0 PL=1
MOVL C00732 V=30.0 PL=1
MOVL C00733 V=30.0 PL=1
MOVL C00734 V=30.0 PL=1
MOVL C00735 V=30.0 PL=1
MOVL C00736 V=30.0 PL=1
MOVL C00737 V=30.0 PL=1
MOVL C00738 V=30.0 PL=1
MOVL C00739 V=130.0 PL=1
MOVL C00740 V=130.0 PL=1
MOVL C00741 V=20.0 PL=1
MOVL C00742 V=130.0 PL=1
MOVL C00743 V=130.0 PL=1
MOVL C00744 V=60.0 PL=1
MOVL C00745 V=60.0 PL=1
MOVL C00746 V=60.0 PL=1
MOVL C00747 V=60.0 PL=1
MOVL C00748 V=130.0 PL=1
MOVL C00749 V=30.0 PL=1
MOVL C00750 V=30.0 PL=1
MOVL C00751 V=30.0 PL=1
MOVL C00752 V=30.0 PL=1
MOVL C00753 V=30.0 PL=1
MOVL C00754 V=30.0 PL=1
MOVL C00755 V=30.0 PL=1
MOVL C00756 V=30.0 PL=1
MOVL C00757 V=130.0 PL=1
MOVL C00758 V=130.0 PL=1
MOVL C00759 V=20.0 PL=1
MOVL C00760 V=130.0 PL=1
MOVL C00761 V=130.0 PL=1
MOVL C00762 V=60.0 PL=1
MOVL C00763 V=60.0 PL=1
MOVL C00764 V=60.0 PL=1
MOVL C00765 V=60.0 PL=1
MOVL C00766 V=130.0 PL=1
MOVL C00767 V=30.0 PL=1
MOVL C00768 V=30.0 PL=1
MOVL C00769 V=30.0 PL=1
MOVL C00770 V=30.0 PL=1
MOVL C00771 V=30.0 PL=1
MOVL C00772 V=30.0 PL=1
MOVL C00773 V=30.0 PL=1
MOVL C00774 V=30.0 PL=1
MOVL C00775 V=130.0 PL=1
MOVL C00776 V=130.0 PL=1
MOVL C00777 V=20.0 PL=1
MOVL C00778 V=130.0 PL=1
MOVL C00779 V=130.0 PL=1
MOVL C00780 V=60.0 PL=1
MOVL C00781 V=60.0 PL=1
MOVL C00782 V=60.0 PL=1
MOVL C00783 V=60.0 PL=1
MOVL C00784 V=130.0 PL=1
MOVL C00785 V=30.0 PL=1
MOVL C00786 V=30.0 PL=1
MOVL C00787 V=30.0 PL=1
MOVL C00788 V=30.0 PL=1
MOVL C00789 V=30.0 PL=1
MOVL C00790 V=30.0 PL=1
MOVL C00791 V=30.0 PL=1
MOVL C00792 V=30.0 PL=1
MOVL C00793 V=130.0 PL=1
MOVL C00794 V=130.0 PL=1
MOVL C00795 V=20.0 PL=1
MOVL C00796 V=130.0 PL=1
MOVL C00797 V=130.0 PL=1
MOVL C00798 V=60.0 PL=1
MOVL C00799 V=60.0 PL=1
MOVL C00800 V=60.0 PL=1
MOVL C00801 V=60.0 PL=1
MOVL C00802 V=130.0 PL=1
MOVL C00803 V=30.0 PL=1
MOVL C00804 V=30.0 PL=1
MOVL C00805 V=30.0 PL=1
MOVL C00806 V=30.0 PL=1
MOVL C00807 V=30.0 PL=1
MOVL C00808 V=30.0 PL=1
MOVL C00809 V=30.0 PL=1
MOVL C00810 V=30.0 PL=1
MOVL C00811 V=130.0 PL=1
MOVL C00812 V=130.0 PL=1
MOVL C00813 V=20.0 PL=1
MOVL C00814 V=130.0 PL=1
MOVL C00815 V=130.0 PL=1
MOVL C00816 V=60.0 PL=1
MOVL C00817 V=60.0 PL=1
MOVL C00818 V=60.0 PL=1
MOVL C00819 V=60.0 PL=1
MOVL C00820 V=130.0 PL=1
MOVL C00821 V=30.0 PL=1
MOVL C00822 V=30.0 PL=1
MOVL C00823 V=30.0 PL=1
MOVL C00824 V=30.0 PL=1
MOVL C00825 V=30.0 PL=1
MOVL C00826 V=30.0 PL=1
MOVL C00827 V=30.0 PL=1
MOVL C00828 V=30.0 PL=1
MOVL C00829 V=130.0 PL=1
MOVL C00830 V=130.0 PL=1
MOVL C00831 V=20.0 PL=1
MOVL C00832 V=130.0 PL=1
MOVL C00833 V=130.0 PL=1
MOVL C00834 V=60.0 PL=1
MOVL C00835 V=60.0 PL=1
MOVL C00836 V=60.0 PL=1
MOVL C00837 V=60.0 PL=1
MOVL C00838 V=130.0 PL=1
MOVL C00839 V=30.0 PL=1
MOVL C00840 V=30.0 PL=1
MOVL C00841 V=30.0 PL=1
MOVL C00842 V=30.0 PL=1
MOVL C00843 V=30.0 PL=1
MOVL C00844 V=30.0 PL=1
MOVL C00845 V=30.0 PL=1
MOVL C00846 V=30.0 PL=1
MOVL C00847 V=130.0 PL=1
MOVL C00848 V=130.0 PL=1
MOVL C00849 V=20.0 PL=1
MOVL C00850 V=130.0 PL=1
MOVL C00851 V=130.0 PL=1
MOVL C00852 V=60.0 PL=1
MOVL C00853 V=60.0 PL=1
MOVL C00854 V=60.0 PL=1
MOVL C00855 V=60.0 PL=1
MOVL C00856 V=130.0 PL=1
MOVL C00857 V=30.0 PL=1
MOVL C00858 V=30.0 PL=1
MOVL C00859 V=30.0 PL=1
MOVL C00860 V=30.0 PL=1
MOVL C00861 V=30.0 PL=1
MOVL C00862 V=30.0 PL=1
MOVL C00863 V=30.0 PL=1
MOVL C00864 V=30.0 PL=1
MOVL C00865 V=130.0 PL=1
MOVL C00866 V=130.0 PL=1
MOVL C00867 V=20.0 PL=1
MOVL C00868 V=130.0 PL=1
MOVL C00869 V=130.0 PL=1
MOVL C00870 V=60.0 PL=1
MOVL C00871 V=60.0 PL=1
MOVL C00872 V=60.0 PL=1
MOVL C00873 V=60.0 PL=1
MOVL C00874 V=130.0 PL=1
MOVL C00875 V=30.0 PL=1
MOVL C00876 V=30.0 PL=1
MOVL C00877 V=30.0 PL=1
MOVL C00878 V=30.0 PL=1
MOVL C00879 V=30.0 PL=1
MOVL C00880 V=30.0 PL=1
MOVL C00881 V=30.0 PL=1
MOVL C00882 V=30.0 PL=1
MOVL C00883 V=130.0 PL=1
MOVL C00884 V=130.0 PL=1
MOVL C00885 V=20.0 PL=1
MOVL C00886 V=130.0 PL=1
MOVL C00887 V=130.0 PL=1
MOVL C00888 V=60.0 PL=1
MOVL C00889 V=60.0 PL=1
MOVL C00890 V=60.0 PL=1
MOVL C00891 V=60.0 PL=1
MOVL C00892 V=130.0 PL=1
MOVL C00893 V=30.0 PL=1
MOVL C00894 V=30.0 PL=1
MOVL C00895 V=30.0 PL=1
MOVL C00896 V=30.0 PL=1
MOVL C00897 V=30.0 PL=1
MOVL C00898 V=30.0 PL=1
MOVL C00899 V=30.0 PL=1
MOVL C00900 V=30.0 PL=1
MOVL C00901 V=130.0 PL=1
MOVL C00902 V=130.0 PL=1
MOVL C00903 V=20.0 PL=1
MOVL C00904 V=130.0 PL=1
MOVL C00905 V=130.0 PL=1
MOVL C00906 V=60.0 PL=1
MOVL C00907 V=60.0 PL=1
MOVL C00908 V=60.0 PL=1
MOVL C00909 V=60.0 PL=1
MOVL C00910 V=130.0 PL=1
MOVL C00911 V=30.0 PL=1
MOVL C00912 V=30.0 PL=1
MOVL C00913 V=30.0 PL=1
MOVL C00914 V=30.0 PL=1
MOVL C00915 V=30.0 PL=1
MOVL C00916 V=30.0 PL=1
MOVL C00917 V=30.0 PL=1
MOVL C00918 V=30.0 PL=1
MOVL C00919 V=130.0 PL=1
MOVL C00920 V=130.0 PL=1
MOVL C00921 V=20.0 PL=1
MOVL C00922 V=130.0 PL=1
MOVL C00923 V=130.0 PL=1
MOVL C00924 V=60.0 PL=1
MOVL C00925 V=60.0 PL=1
MOVL C00926 V=60.0 PL=1
MOVL C00927 V=60.0 PL=1
MOVL C00928 V=130.0 PL=1
MOVL C00929 V=30.0 PL=1
MOVL C00930 V=30.0 PL=1
MOVL C00931 V=30.0 PL=1
MOVL C00932 V=30.0 PL=1
MOVL C00933 V=30.0 PL=1
MOVL C00934 V=30.0 PL=1
MOVL C00935 V=30.0 PL=1
MOVL C00936 V=30.0 PL=1
MOVL C00937 V=130.0 PL=1
MOVL C00938 V=130.0 PL=1
MOVL C00939 V=20.0 PL=1
MOVL C00940 V=130.0 PL=1
MOVL C00941 V=130.0 PL=1
MOVL C00942 V=60.0 PL=1
MOVL C00943 V=60.0 PL=1
MOVL C00944 V=60.0 PL=1
MOVL C00945 V=60.0 PL=1
MOVL C00946 V=130.0 PL=1
MOVL C00947 V=30.0 PL=1
MOVL C00948 V=30.0 PL=1
MOVL C00949 V=30.0 PL=1
MOVL C00950 V=30.0 PL=1
MOVL C00951 V=30.0 PL=1
MOVL C00952 V=30.0 PL=1
MOVL C00953 V=30.0 PL=1
MOVL C00954 V=30.0 PL=1
MOVL C00955 V=130.0 PL=1
MOVL C00956 V=130.0 PL=1
MOVL C00957 V=20.0 PL=1
MOVL C00958 V=130.0 PL=1
MOVL C00959 V=130.0 PL=1
MOVL C00960 V=60.0 PL=1
MOVL C00961 V=60.0 PL=1
MOVL C00962 V=60.0 PL=1
MOVL C00963 V=60.0 PL=1
MOVL C00964 V=130.0 PL=1
MOVL C00965 V=30.0 PL=1
MOVL C00966 V=30.0 PL=1
MOVL C00967 V=30.0 PL=1
MOVL C00968 V=30.0 PL=1
MOVL C00969 V=30.0 PL=1
MOVL C00970 V=30.0 PL=1
MOVL C00971 V=30.0 PL=1
MOVL C00972 V=30.0 PL=1
MOVL C00973 V=130.0 PL=1
MOVL C00974 V=130.0 PL=1
MOVL C00975 V=20.0 PL=1
MOVL C00976 V=130.0 PL=1
MOVL C00977 V=130.0 PL=1
MOVL C00978 V=60.0 PL=1
MOVL C00979 V=60.0 PL=1
MOVL C00980 V=60.0 PL=1
MOVL C00981 V=60.0 PL=1
MOVL C00982 V=130.0 PL=1
MOVL C00983 V=30.0 PL=1
MOVL C00984 V=30.0 PL=1
MOVL C00985 V=30.0 PL=1
MOVL C00986 V=30.0 PL=1
MOVL C00987 V=30.0 PL=1
MOVL C00988 V=30.0 PL=1
MOVL C00989 V=30.0 PL=1
MOVL C00990 V=30.0 PL=1
MOVL C00991 V=130.0 PL=1
MOVL C00992 V=130.0 PL=1
MOVL C00993 V=20.0 PL=1
MOVL C00994 V=130.0 PL=1
MOVL C00995 V=130.0 PL=1
MOVL C00996 V=60.0 PL=1
MOVL C00997 V=60.0 PL=1
MOVL C00998 V=60.0 PL=1
MOVL C00999 V=60.0 PL=1
MOVL C01000 V=130.0 PL=1
MOVL C01001 V=30.0 PL=1
MOVL C01002 V=30.0 PL=1
MOVL C01003 V=30.0 PL=1
MOVL C01004 V=30.0 PL=1
MOVL C01005 V=30.0 PL=1
MOVL C01006 V=30.0 PL=1
MOVL C01007 V=30.0 PL=1
MOVL C01008 V=30.0 PL=1
MOVL C01009 V=130.0 PL=1
MOVL C01010 V=130.0 PL=1
MOVL C01011 V=20.0 PL=1
MOVL C01012 V=130.0 PL=1
MOVL C01013 V=130.0 PL=1
MOVL C01014 V=60.0 PL=1
MOVL C01015 V=60.0 PL=1
MOVL C01016 V=60.0 PL=1
MOVL C01017 V=60.0 PL=1
MOVL C01018 V=130.0 PL=1
MOVL C01019 V=30.0 PL=1
MOVL C01020 V=30.0 PL=1
MOVL C01021 V=30.0 PL=1
MOVL C01022 V=30.0 PL=1
MOVL C01023 V=30.0 PL=1
MOVL C01024 V=30.0 PL=1
MOVL C01025 V=30.0 PL=1
MOVL C01026 V=30.0 PL=1
MOVL C01027 V=130.0 PL=1
MOVL C01028 V=130.0 PL=1
MOVL C01029 V=20.0 PL=1
MOVL C01030 V=130.0 PL=1
MOVL C01031 V=130.0 PL=1
MOVL C01032 V=60.0 PL=1
MOVL C01033 V=60.0 PL=1
MOVL C01034 V=60.0 PL=1
MOVL C01035 V=60.0 PL=1
MOVL C01036 V=130.0 PL=1
MOVL C01037 V=30.0 PL=1
MOVL C01038 V=30.0 PL=1
MOVL C01039 V=30.0 PL=1
MOVL C01040 V=30.0 PL=1
MOVL C01041 V=30.0 PL=1
MOVL C01042 V=30.0 PL=1
MOVL C01043 V=30.0 PL=1
MOVL C01044 V=30.0 PL=1
MOVL C01045 V=130.0 PL=1
MOVL C01046 V=130.0 PL=1
MOVL C01047 V=20.0 PL=1
MOVL C01048 V=130.0 PL=1
MOVL C01049 V=130.0 PL=1
MOVL C01050 V=60.0 PL=1
MOVL C01051 V=60.0 PL=1
MOVL C01052 V=60.0 PL=1
MOVL C01053 V=60.0 PL=1
MOVL C01054 V=130.0 PL=1
MOVL C01055 V=30.0 PL=1
MOVL C01056 V=30.0 PL=1
MOVL C01057 V=30.0 PL=1
MOVL C01058 V=30.0 PL=1
MOVL C01059 V=30.0 PL=1
MOVL C01060 V=30.0 PL=1
MOVL C01061 V=30.0 PL=1
MOVL C01062 V=30.0 PL=1
MOVL C01063 V=130.0 PL=1
MOVL C01064 V=130.0 PL=1
MOVL C01065 V=20.0 PL=1
MOVL C01066 V=130.0 PL=1
MOVL C01067 V=130.0 PL=1
MOVL C01068 V=60.0 PL=1
MOVL C01069 V=60.0 PL=1
MOVL C01070 V=60.0 PL=1
MOVL C01071 V=60.0 PL=1
MOVL C01072 V=130.0 PL=1
MOVL C01073 V=30.0 PL=1
MOVL C01074 V=30.0 PL=1
MOVL C01075 V=30.0 PL=1
MOVL C01076 V=30.0 PL=1
MOVL C01077 V=30.0 PL=1
MOVL C01078 V=30.0 PL=1
MOVL C01079 V=30.0 PL=1
MOVL C01080 V=30.0 PL=1
MOVL C01081 V=130.0 PL=1
MOVL C01082 V=130.0 PL=1
MOVL C01083 V=20.0 PL=1
MOVL C01084 V=130.0 PL=1
MOVL C01085 V=130.0 PL=1
MOVL C01086 V=60.0 PL=1
MOVL C01087 V=60.0 PL=1
MOVL C01088 V=60.0 PL=1
MOVL C01089 V=60.0 PL=1
MOVL C01090 V=130.0 PL=1
MOVL C01091 V=30.0 PL=1
MOVL C01092 V=30.0 PL=1
MOVL C01093 V=30.0 PL=1
MOVL C01094 V=30.0 PL=1
MOVL C01095 V=30.0 PL=1
MOVL C01096 V=30.0 PL=1
MOVL C01097 V=30.0 PL=1
MOVL C01098 V=30.0 PL=1
MOVL C01099 V=130.0 PL=1
MOVL C01100 V=130.0 PL=1
MOVL C01101 V=20.0 PL=1
MOVL C01102 V=130.0 PL=1
MOVL C01103 V=130.0 PL=1
MOVL C01104 V=60.0 PL=1
MOVL C01105 V=60.0 PL=1
MOVL C01106 V=60.0 PL=1
MOVL C01107 V=60.0 PL=1
MOVL C01108 V=130.0 PL=1
MOVL C01109 V=30.0 PL=1
MOVL C01110 V=30.0 PL=1
MOVL C01111 V=30.0 PL=1
MOVL C01112 V=30.0 PL=1
MOVL C01113 V=30.0 PL=1
MOVL C01114 V=30.0 PL=1
MOVL C01115 V=30.0 PL=1
MOVL C01116 V=30.0 PL=1
MOVL C01117 V=130.0 PL=1
MOVL C01118 V=130.0 PL=1
MOVL C01119 V=20.0 PL=1
MOVL C01120 V=130.0 PL=1
MOVL C01121 V=130.0 PL=1
MOVL C01122 V=60.0 PL=1
MOVL C01123 V=60.0 PL=1
MOVL C01124 V=60.0 PL=1
MOVL C01125 V=60.0 PL=1
MOVL C01126 V=130.0 PL=1
MOVL C01127 V=30.0 PL=1
MOVL C01128 V=30.0 PL=1
MOVL C01129 V=30.0 PL=1
MOVL C01130 V=30.0 PL=1
MOVL C01131 V=30.0 PL=1
MOVL C01132 V=30.0 PL=1
MOVL C01133 V=30.0 PL=1
MOVL C01134 V=30.0 PL=1
MOVL C01135 V=130.0 PL=1
MOVL C01136 V=130.0 PL=1
MOVL C01137 V=20.0 PL=1
MOVL C01138 V=130.0 PL=1
MOVL C01139 V=130.0 PL=1
MOVL C01140 V=60.0 PL=1
MOVL C01141 V=60.0 PL=1
MOVL C01142 V=60.0 PL=1
MOVL C01143 V=60.0 PL=1
MOVL C01144 V=130.0 PL=1
MOVL C01145 V=30.0 PL=1
MOVL C01146 V=30.0 PL=1
MOVL C01147 V=30.0 PL=1
MOVL C01148 V=30.0 PL=1
MOVL C01149 V=30.0 PL=1
MOVL C01150 V=30.0 PL=1
MOVL C01151 V=30.0 PL=1
MOVL C01152 V=30.0 PL=1
MOVL C01153 V=130.0 PL=1
MOVL C01154 V=130.0 PL=1
MOVL C01155 V=20.0 PL=1
MOVL C01156 V=130.0 PL=1
MOVL C01157 V=130.0 PL=1
MOVL C01158 V=60.0 PL=1
MOVL C01159 V=60.0 PL=1
MOVL C01160 V=60.0 PL=1
MOVL C01161 V=60.0 PL=1
END
